			IF (tmrHorEntryNotPresent.q AND I_HOR_DnStream_Cv_Full) OR
				mc.DryRun THEN
				TimeoutTrigger 					:= FALSE;
				Station.RunStep	:= Station.RunStep + 10;
			END_IF

	40 : 	(************* Carton Send to Exit Conveyor  ****************)
			Station.Status 		:= '40: Carton Send to Exit Conveyor';
			Station.StatusInt	:= 354;
			
			IF NOT A_HOR_LC_Muting THEN
				HOR_BotCv_Mtr_Var.In_AutoON 			:= 	FALSE;
				HOR_TopCv_Mtr_Var.In_AutoON 			:= 	FALSE;


			(*	Case Counter *)				
					Statistic_CurShift_CaseProduce		:= Statistic_CurShift_CaseProduce + 1;
					Statistic_Total_CaseProduce			:= Statistic_Total_CaseProduce	+1;
					Statistic_Man_Total_CaseProduce		:= Statistic_Man_Total_CaseProduce +1;
					
			(* Update Statistic *)
			IF NOT mc.DryRun THEN
				IF NOT TapeReel_ActivatedL OR  W_HOR_TapeLRefill THEN
					Statistic_Current.RejectLeftTape	:= Statistic_Current.RejectLeftTape + 1;
					Statistic_Manual.RejectLeftTape		:= Statistic_Manual.RejectLeftTape + 1;
					Statistic_Total.RejectLeftTape		:= Statistic_Total.RejectLeftTape + 1;					
					E_CartonTapingErrL					:= TRUE;	
					Exit_Case_NG 						:= TRUE;
				
					
				ELSIF NOT TapeReel_ActivatedR OR W_HOR_TapeRRefill THEN
					Statistic_Current.RejectRightTape	:= Statistic_Current.RejectRightTape + 1;
					Statistic_Manual.RejectRightTape	:= Statistic_Manual.RejectRightTape + 1;
					Statistic_Total.RejectRightTape		:= Statistic_Total.RejectRightTape + 1;
					E_CartonTapingErrR					:= TRUE;	
					Exit_Case_NG 						:= TRUE;

					
				ELSIF 	H_CartonWeight < (CurrRecipe.rWeightTarget - CurrRecipe.rWeightTol) AND Cfg_EnbWeightCheck THEN
					Statistic_Current.RejectUnderWeight	:= Statistic_Current.RejectUnderWeight	+ 1;
					Statistic_Manual.RejectUnderWeight	:= Statistic_Manual.RejectUnderWeight	+ 1;
					Statistic_Total.RejectUnderWeight	:= Statistic_Total.RejectUnderWeight	+ 1;
					Weight_Fail_Counter					:= Weight_Fail_Counter +1;
					Exit_Case_NG 						:= TRUE;
					
					
				ELSIF 	H_CartonWeight > (CurrRecipe.rWeightTarget + CurrRecipe.rWeightTol) AND Cfg_EnbWeightCheck THEN
					Statistic_Current.RejectOverWeight	:= Statistic_Current.RejectOverWeight + 1;
					Statistic_Manual.RejectOverWeight	:= Statistic_Manual.RejectOverWeight + 1;
					Statistic_Total.RejectOverWeight	:= Statistic_Total.RejectOverWeight + 1;
					Weight_Fail_Counter					:= Weight_Fail_Counter +1;
					Exit_Case_NG 						:= TRUE;

			
				ELSE
					Statistic_Current.GoodCase			:= Statistic_Current.GoodCase + 1;	
					Statistic_Manual.GoodCase			:= Statistic_Manual.GoodCase + 1;	
					Statistic_Total.GoodCase			:= Statistic_Total.GoodCase + 1;	
					Exit_Case_Good 						:= TRUE;
					Weight_Fail_Counter					:= 0;


				END_IF
				
			ELSE
					Statistic_Manual.GoodCase			:= Statistic_Manual.GoodCase + 1;
					Weight_Fail_Counter					:= 0;

			END_IF		
								
				Station.RunStep	:= Station.RunStep + 10;
			END_IF
	
	50: (************* Tilt In conveyor waiting for carton in position ****************)
			Station.Status 		:= '50: Tilt Conveyor Waiting For Carton In Position';
			
			HOR_Tilt_In_Mtr_Var.In_AutoON	:= TRUE;
			HOR_Tilt_Out_Mtr_Var.In_AutoON	:= TRUE;

			IF (TiltInCv_InPosDly.Q OR mc.DryRun) AND NOT I_HOR_Tilt_Out_Cv_Present  THEN	
				Station.RunStep	:= Station.RunStep + 10;
			END_IF	
				
	60: (************* Tilt Unit Tilt to Tilt Out Conveyor ****************)
			Station.Status 		:= '60: Tilt Unit Tilt Carton To Out Conveyor';
			
			EX_Tilt_Srv_Var.In_PosCmd := 85.0;
			EX_Tilt_Srv_Var.In_VelCmd := 100;
			EX_Tilt_Srv_Var.In_MoveAbs := TRUE; 
	
			IF fcComparePos(CurrPos:= EX_Tilt_Srv_Var.Out_CurrPos, TargetPos:= EX_Tilt_Srv_Var.In_PosCmd, Tolerance := 0.5) THEN
				EX_Tilt_Srv_Var.In_MoveAbs := FALSE; 
				Station.RunStep	:= 10000;
			END_IF
			(*temporarily disable referencing*)
	
	70: (************* Tilt Unit Start Seaching for Sensor ****************)
			Station.Status 		:= '70: Tilt Unit Searching for Home Sensor';
		
			EX_Tilt_Srv_Var.In_SetAbsRef	:= TRUE;
	
			IF NOT EX_Tilt_Srv_Var.Out_Referenced THEN
				Station.RunStep	:= Station.RunStep + 10;
			END_IF
	80: (************* Tilt Unit Waiting for Home Sensor ****************)	
			Station.Status 		:= '80: Tilt Unit Waiting for Homing Complete';
			
			HOR_Tilt_In_Mtr_Var.In_AutoON		:= FALSE;
	
	
			IF  EX_Tilt_Srv_Var.Out_Referenced THEN
				EX_Tilt_Srv_Var.In_SetAbsRef	:= FALSE;
				Station.RunStep					:= 1000;
			END_IF
			
	1000 : 	(************* Process Done ****************)
			Station.Status 		:= '1000: Process Done';	
			Station.StatusInt	:= 499;
			M_StepRun 			:= FALSE;
			HMI.T_OneCycleRun 	:= FALSE;			
			Station.RunStep 	:= 0;
			H_ER_CtnGlueDone	:= FALSE;
			H_HOR_CtnWeightOK	:= FALSE;
			TimeoutTrigger 		:= FALSE;
	END_CASE

(* Tilt Out Conveyor Stop *)
IF TiltOutCv_StopDly.Q	THEN
	HOR_Tilt_Out_Mtr_Var.In_AutoON		:= FALSE;
END_IF

	

ELSE
	Station.RunStep := 0;
	
	IF Station.MajorFault OR Station.MinorFault THEN
		Station.Status 		:= 'Station Error';
		Station.StatusInt	:= 4;
	ELSIF Station.Origin THEN
		Station.Status 		:= 'Station In Origin';
		Station.StatusInt	:= 5;
	ELSIF NOT Station.OriginSchRun AND NOT MC.OriginSchRun THEN
		Station.Status 		:= 'Station Not In Origin';
		Station.StatusInt	:= 6;
	END_IF
END_IF

Station.Running := (Station.RunStep>0) OR (sc[4].RunStep >0) ;

END_PROGRAM

// ---- POUs/Horizontal/HOR_Origin.TcPOU
PROGRAM HOR_Origin
VAR_IN_OUT
	Station		:structStationCtrl;
END_VAR
VAR
	HOR_WA_Origin		:BOOL;
	pls_OriginSchRun	:R_trig;
	Timeout				:Ton;
	TmrCartonExit		:Ton;
	TimeoutTrigger		:BOOL;
	TimeoutSetting		:TIME;
	tmr_FullSensorDly	:TON;
	tmr_MtrStopped		:ton;
		
END_VAR

(**************************************************************************************************************)
(* Station Width Adjust in Origin Condition *)
(**************************************************************************************************************)
HOR_WA_Origin := 	TRUE ;

(**************************************************************************************************************)
(* Station Origin Condition *)
(**************************************************************************************************************)

Station.Origin 	:=	(
					(NOT I_HOR_Entry_Cv_Present OR H_ER_CtnGlueDone) AND
					HOR_BotCv_Mtr_Var.S_InvRdy AND
					HOR_TopCv_Mtr_Var.S_InvRdy AND
					HOR_WA_Origin AND
					EX_Tilt_Srv_Var.Out_Referenced AND
					tmr_MtrStopped.Q and
					Station.OriginRunStep =0)OR
					Station.Bypass;
					 		
(**************************************************************************************************************)
(* Individual Station Origin Run Trigger *)
(**************************************************************************************************************)
IF MC.ManualMode AND NOT Station.Origin AND NOT (Station.MajorFault OR Station.MinorFault OR MC.Trouble OR MC.StopPressed )  THEN
	IF Station.T_OriginSearch THEN
		Station.OriginSchRun  := TRUE;
	END_IF;
ELSE
	Station.OriginSchRun := FALSE;
	HOR.T_OriginSearch := FALSE;
END_IF;

(**************************************************************************************************************)
(* Station Origin Step *)
(**************************************************************************************************************)

Timeout(IN:=TimeoutTrigger, PT:=TimeoutSetting);
IF Timeout.Q THEN
	TimeoutTrigger := FALSE;
END_IF

pls_OriginSchRun(CLK:= (MC.OriginSchRun OR Station.OriginSchRun));
TmrCartonExit (in:= NOT I_HOR_DnStream_Cv_Full AND NOT I_HOR_Entry_Cv_Present  AND (Station.OriginRunStep = 30), pt:=T#10S);
tmr_FullSensorDly (IN:= (Station.OriginRunStep >= 30) AND I_HOR_DnStream_Cv_Full, PT:= T#3S);
tmr_MtrStopped( IN:= NOT HOR_BotCv_Mtr_Var.S_Running AND NOT HOR_TopCv_Mtr_Var.S_Running , pt:= T#2S);

IF (MC.OriginSchRun OR Station.OriginSchRun) AND NOT Station.Bypass  THEN
	CASE Station.OriginRunStep OF

	0 : 	(************* Ready To Run ****************)
			IF NOT Station.Origin AND pls_OriginSchRun.Q THEN
				Station.OriginRunStep := Station.OriginRunStep+10;	
			END_IF

	10	:	(************* Clear Tilt In and Tilt Out Conveyor ****************)
			Station.Status := 'Org10: Tilt Conveyor In and Out Run';
			
			HOR_Tilt_In_Mtr_Var.In_OrgOn	:= TRUE;
			HOR_Tilt_Out_Mtr_Var.In_OrgOn	:= TRUE;

			IF NOT I_HOR_Tilt_Out_Cv_Present THEN
				Station.OriginRunStep := Station.OriginRunStep+10;
			END_IF
			
	20:		(************ Tilt Unit Origin **********************)
			Station.Status := 'Org20: Tilt Servo Start to Home';
			
			EX_Tilt_Srv_Var.In_SetAbsRef	:= TRUE;
			
			IF NOT EX_Tilt_Srv_Var.Out_Referenced THEN
				Station.OriginRunStep	:= Station.OriginRunStep + 10;
			END_IF
	
	30: (***************** Waiting for Tilt Unit Origin Done ************)
			Station.Status := 'Org30: Tilt Servo Homing';
		
			IF  EX_Tilt_Srv_Var.Out_Referenced THEN
				EX_Tilt_Srv_Var.In_SetAbsRef	:= FALSE;
				Station.OriginRunStep	:= Station.OriginRunStep + 10;
			END_IF
		
	40 : 	(************* Cek Carton On Conveyor ****************)
			Station.Status := 'Org40: Cek Carton On Conveyor';
			HOR_BotCv_Mtr_Var.In_OrgOn	:= TRUE;
			HOR_TopCv_Mtr_Var.In_OrgOn	:= TRUE;
			EX_StpCylR_Var.In_OrgHome	:= TRUE;
			EX_StpCylL_Var.In_OrgHome	:= TRUE;
			
			IF I_HOR_Entry_Cv_Present THEN
				Station.Status := 'Org10: Top and Bottom Motor Run';
			ELSE
				Station.OriginRunStep := Station.OriginRunStep+10;
			END_IF
	
	50 : 	(************* Carton Send to Exit Conveyor  ****************)
			Station.Status 		:= 'Org50: Carton Send to Exit Conveyor';
			
			
			IF NOT I_HOR_Entry_Cv_Present THEN
				Station.OriginRunStep	:= Station.OriginRunStep + 10;
			END_IF

	60 : 	(************* Carton Send to Exit Conveyor  ****************)
			Station.Status 		:= 'Org60: Carton Send to Exit Conveyor';
			Station.StatusInt	:= 354;
			
			H_ER_CtnRdyForGlue	:=FALSE;
			H_ER_CtnGlueDone	:=FALSE;
			H_ER_CtnWeightOK	:=FALSE;				

			IF  tmr_FullSensorDly.Q OR TmrCartonExit.q THEN

				EX_StpCylR_Var.In_Orgwork	:= TRUE;
				EX_StpCylL_Var.In_Orgwork	:= TRUE;
				EX_StpCylR_Var.In_OrgHome	:= FALSE;
				EX_StpCylL_Var.In_OrgHome	:= FALSE;
				Station.OriginRunStep 		:= 40;
			END_IF

	70:	(******************** Make sure Conveyor is stopped **********************)
				HOR_BotCv_Mtr_Var.In_OrgOn 		:= FALSE;
				HOR_TopCv_Mtr_Var.In_OrgOn		:= FALSE;
				HOR_BotCv_Mtr_Var.T_ManOn 		:= FALSE;
				HOR_TopCv_Mtr_Var.T_ManOn		:= FALSE;	
				HOR_Tilt_In_Mtr_Var.In_OrgOn	:= FALSE;
				HOR_Tilt_Out_Mtr_Var.In_OrgOn	:= FALSE;				
			
		IF  tmr_MtrStopped.Q THEN
				Station.OriginRunStep 		:= 0;
			END_IF
		
	END_CASE

ELSE

	Station.OriginRunStep := 0;	

	
END_IF

END_PROGRAM

// ---- POUs/Horizontal/Option_90Deg_Conv.TcPOU
PROGRAM Option_90Deg_Conv
VAR
	bEnable			:BOOL;
	Full_Timer_ON	: TON;
	Clear_Timer_ON	: tOF;
	
END_VAR

bEnable := NOT MC.Trouble;
Full_Timer_ON	(IN:= I_HOR_DnStream_Cv_Full , PT:= T#2S);
Clear_Timer_ON	(IN:= I_HOR_90Deg_Full_PE, PT:= T#3S);

EX_Deg_Cyl_Var.In_HomeXLock := TRUE;
EX_Deg_Cyl_Var.In_WorkXLock := TRUE;

EX_90Deg_Cyl(				
	IN_CylName		:='TILT CV CYLINDER', 	
	In_Enable		:= Cfg_Exit90DegConv, 	
	In_Reset		:= MC.ResetPressed, 	
	In_WorkRS		:= I_HOR_90Deg_Tilt_Cly_Up, 	
	In_HomeRS		:= I_HOR_90Deg_Tilt_Cly_Dn, 	
	In_WorkTON		:= T#100MS, 	
	In_HomeTON		:= T#10MS, 	
	in_Timeout		:= T#5S, 	
	Out_WorkSV		=> O_HOR_90Deg_Cyl_Up, 	
	Out_HomeSV		=> O_HOR_90Deg_Cyl_Dn, 	
	CylVar			:= EX_Deg_Cyl_Var,
	Station			:= SC[6]);
	
(*	Control Condition	*)
IF 	SC[6].AutoRun			AND
	Full_Timer_ON.Q	AND
	not Clear_Timer_ON.q THEN
	EX_Deg_Cyl_Var.In_AutoWork	:= TRUE;
	EX_Deg_Cyl_Var.In_AutoHome	:= FALSE;
ELSE
	EX_Deg_Cyl_Var.In_AutoWork	:= FALSE;
	EX_Deg_Cyl_Var.In_AutoHome	:= TRUE;
END_IF

END_PROGRAM

// ---- POUs/Horizontal/HOR_Servo_Output.TcPOU
PROGRAM HOR_Servo_Output
VAR
	Reset:BOOL;
	bEnable:BOOL;
	plsStopMove: R_trig;
	debugcode: INT;
	debugcode2: INT;
END_VAR

IF (MC.AutoMode OR SC[6].M_Step) THEN
	EX_Tilt_Srv_Var.In_ServoOn := TRUE;
END_IF

IF HOR.OriginSchRun OR MC.OriginSchRun OR mc.AutoMode OR (mc.ResetPressed AND NOT mc.Trouble) THEN
	EX_Tilt_Srv_Var.In_ServoOn := TRUE;
END_IF

bEnable := NOT (SC[6].MajorFault OR MC.Trouble);

EX_Tilt_Srv_Var.In_MoveXLock := TRUE ;
EX_Tilt_Srv_Input.wSignalstatuswort.13	:= TRUE;
EX_Tilt_Srv_Input.wSignalstatuswort.14	:= TRUE;


EX_Tilt_Srv_Drive(
	In_Enable:= bEnable, 
	In_Reset := MC.ResetPressed,
	In_AbsEncoder:= FALSE, 
	In_DriveInput:= EX_Tilt_Srv_Input, 
	In_CommState:= EX_Tilt_Srv_State, 
	Out_DriveOutput=> EX_Tilt_Srv_Output, 
	Out_DriveFeedRateOverride=> , 
	DriveVar:= EX_Tilt_Srv_Var,
	Station			:= SC[6]);
	
IF mc.ManualMode THEN	
	EX_Tilt_Srv_Feedrate := 10000;
ELSE
	EX_Tilt_Srv_Feedrate :=    INT_TO_UINT(hmi.V_MachineSpeed * 100);
END_IF

END_PROGRAM

// ---- POUs/Horizontal/HOR_Motor_Output.TcPOU
PROGRAM HOR_Motor_Output
VAR
	Reset:BOOL;
	bEnable: BOOL;
	bManualReject	:BOOL;
	tmrManualReject	:Ton;
	bManualRejectNeg	:R_trig;
	
	
END_VAR

(******************** Error Stop ***********************)
IF E_Top_Conv_Jam or E_Bottom_Conv_Jam  THEN
	HOR_BotCv_Mtr_Var.E_OnErr	:= TRUE;
	HOR_TopCv_Mtr_Var.E_OnErr	:= TRUE;
END_IF
(********************************************************)

bEnable := NOT MC.Trouble AND Cfg_HorizontalExit;
HOR_BotCv_Mtr_Var.In_SpeedSel :=3;
HOR_BotCv_Mtr_Var.In_MoveXLock := TRUE;

HOR_BotCv_Mtr(
	IN_DevName:= 'HORIZON. BOTTOM CV', 
	In_Enable:= bEnable, 
	In_Reset:= MC.ResetPressed, 
	In_InvRdy := I_HOR_BotCv_InvRdy, 
	Out_InvRun => O_HOR_BotCv_Mtr_Run, 
	Out_InvDirc => O_HOR_BotCv_Mtr_Dirc, 
	Out_InvSpdBit0 => O_HOR_BotCv_Mtr_Spd1, 
	Out_InvSpdBit1 => O_HOR_BotCv_Mtr_Spd2,
	MotorVar:= HOR_BotCv_Mtr_Var,
	Station			:= SC[6]);


HOR_TopCv_Mtr_Var.In_MoveXLock := TRUE;
HOR_TopCv_Mtr_Var.In_SpeedSel :=3;
HOR_TopCv_Mtr(
	IN_DevName:= 'HORIZON. TOP CV', 
	In_Enable:= bEnable, 
	In_Reset:= MC.ResetPressed, 
	In_InvRdy := I_HOR_TopCv_InvRdy, 
	Out_InvRun => O_HOR_TopCv_Mtr_Run, 
	Out_InvDirc => O_HOR_TopCv_Mtr_Dirc, 
	Out_InvSpdBit0 => O_HOR_TopCv_Mtr_Spd1, 
	Out_InvSpdBit1 => O_HOR_TopCv_Mtr_Spd2,
	MotorVar:= HOR_TopCv_Mtr_Var,
	Station			:= SC[6]);


(* Reject Carton Manually *)	
tmrManualReject		(in:= bManualReject, pt:= T#10S);
bManualRejectNeg	( CLK := tmrManualReject.Q);

IF NOT tmrManualReject.Q AND bManualReject THEN
	HOR_TopCv_Mtr_Var.T_ManOn	:= TRUE;
	HOR_TopCv_Mtr_Var.T_ManOff	:= FALSE;
	WT_Mtr_Var.T_ManOn			:= TRUE;
	WT_Mtr_Var.T_ManOff			:= FALSE;
	HOR_BotCv_Mtr_Var.T_ManOn	:= TRUE;
	HOR_BotCv_Mtr_Var.T_ManOff	:= FALSE;	
	EX_FlapHoldL_Cyl_Var.T_ManHome	:= TRUE;
	EX_FlapHoldL_Cyl_Var.T_ManWork	:= FALSE;
	EX_FlapHoldR_Cyl_Var.T_ManHome	:= TRUE;
	EX_FlapHoldR_Cyl_Var.T_ManWork	:= FALSE;	
	Ex_SquarenessCylL_Var.T_ManHome	:= TRUE;
	Ex_SquarenessCylL_Var.T_ManWork	:= FALSE;
	Ex_SquarenessCylR_Var.T_ManHome	:= TRUE;
	Ex_SquarenessCylR_Var.T_ManWork	:= FALSE;	
	EX_StpCylL_Var.T_ManHome		:= TRUE;
	EX_StpCylL_Var.T_ManWork		:= FALSE;
	EX_StpCylR_Var.T_ManHome		:= TRUE;
	EX_StpCylR_Var.T_ManWork		:= FALSE;	
	
	IF 	H_ER_CtnRdyForGlue OR H_ER_CtnGlueDone OR H_ER_CtnWeightOK THEN
		Statistic_Current.RejectCaseRemoved	:= Statistic_Current.RejectCaseRemoved + 1;
		Statistic_Manual.RejectCaseRemoved	:= Statistic_Manual.RejectCaseRemoved + 1;
		Statistic_Total.RejectCaseRemoved	:= Statistic_Total.RejectCaseRemoved + 1;
	END_IF
	
	HMI.T_ClearExitMem			:= TRUE;	
END_IF

IF bManualRejectNeg.Q  THEN
	HOR_TopCv_Mtr_Var.T_ManOn	:= FALSE;
	WT_Mtr_Var.T_ManOn			:= FALSE;
	HOR_BotCv_Mtr_Var.T_ManOn	:= FALSE;
	bManualReject				:= FALSE;
	HOR_TopCv_Mtr_Var.T_ManOff	:= TRUE;
	WT_Mtr_Var.T_ManOff			:= TRUE;
	HOR_BotCv_Mtr_Var.T_ManOff	:= TRUE;	
	HMI.T_ClearExitMem			:= FALSE;		
END_IF
(* Tilt In Conveyor *)
HOR_Tilt_In_Mtr_Var.In_MoveXLock := TRUE;
	
HOR_Tilt_In_Mtr(
	IN_DevName:= 'Tilt In CV', 
	In_Enable:= bEnable, 
	In_Reset:= MC.ResetPressed, 
	In_StarterOK:= TRUE, 
	Out_MotorOn=> O_HOR_TiltCV1_On, 
	MotorVar:= HOR_Tilt_In_Mtr_Var,
	Station			:= SC[6]);

(* Tilt Out Conveyor *)
HOR_Tilt_Out_Mtr_Var.In_MoveXLock := TRUE;
	
HOR_Tilt_Out_Mtr(
	IN_DevName:= 'Tilt Out CV', 
	In_Enable:= bEnable, 
	In_Reset:= MC.ResetPressed, 
	In_StarterOK:= TRUE, 
	Out_MotorOn=> O_HOR_TiltCV2_On, 
	MotorVar:= HOR_Tilt_Out_Mtr_Var,
	Station			:= SC[6]);

END_PROGRAM

// ---- POUs/MC/Track_and_Trace.TcPOU
PROGRAM Track_and_Trace
VAR
tmr_TnT_CrossPushToCase		: Tof;
tmr_TnT_CrossPushForward	: Tof;
tmr_TnT_CaseIndex			: Tof;	
tmr_TnT_GoodCaseDischarge	: Tof;


END_VAR

(* Case Format *)
(* 2.2.1	Case format *)
(* (for differentiation between 5000 and 10000 cases 0 for 5000 and 1 for 10000)*)
IF CurrRecipe.iStackY = 2 THEN
		O_TnT_CaseFormat	:= TRUE;
	ELSE
		O_TnT_CaseFormat	:= FALSE;	
END_IF

(* Cross push to case initiated *)
(* 2.2.2	Cross push to case initiated (signal to go high as cross push starts) *)
tmr_TnT_CrossPushToCase (IN:= SC[2].RunStep	= 10 , PT:= T#1S);
O_TnT_CrossPushToCase	:= tmr_TnT_CrossPushToCase.Q;

(* Cross Push Fully Forward *)
(* 2.2.3	Cross push fully forward (Outers pushed into case- signal to go high)*)
tmr_TnT_CrossPushForward (IN:= SC[2].RunStep	= 110 , PT:= T#1S);
O_TnT_CrossPushForward	:= tmr_TnT_CrossPushForward.Q;

(* Case Index *)
(* 2.2.4	Case index (as machine indexes signal to go high at start of index)*)
tmr_TnT_CaseIndex	(IN:= SC[3].RunStep	= 30 , PT:= T#1S);
O_TnT_CaseIndex			:= tmr_TnT_CaseIndex.Q;

(* Good Case Discharge *)
(* 2.2.5	Good case discharged (i.e. signal high if case is not to be rejected – on as case exits machine)*)
tmr_TnT_GoodCaseDischarge	(IN:= Exit_Case_Good , PT:= T#1S);
O_TnT_GoodCaseDischarge		:= tmr_TnT_GoodCaseDischarge.Q;

END_PROGRAM

// ---- POUs/MC/Memory_Handling.TcPOU
PROGRAM Memory_Handling
VAR
	plsMemoryReset: R_trig;
	plsPurgeErectorCaseOff: R_trig;
	T_ManPurge: INT;
	tmrPurgeErectorCase:tof;
END_VAR

plsMemoryReset(CLK:=MC.DryRun);

IF plsMemoryReset.Q OR HMI.T_ClearAllMem OR MC_WA_Run THEN
	H_CO_StkRdyForXPush:=FALSE;
	H_CO_StkRdyForYPush:=FALSE;	
	H_ER_CtnRdyForPushIn:=FALSE;
	H_ER_CtnPushInDone:=FALSE;
	H_ER_CtnSideFlapDone:=FALSE;
	H_ER_CtnRdyForGlue:=FALSE;
	H_ER_CtnGlueDone:=FALSE;
	H_ER_CtnWeightOK:=FALSE;
	H_EL_CtnTapeDone:=FALSE;
	H_EL_CtnWeightOK:=FALSE;
	H_CO_Bdl_StkY_Count := 0;
	H_CO_Bdl_StkZ_Count := 0;
END_IF

IF HMI.T_ClearCollatorMem THEN
	H_CO_StkRdyForXPush:=FALSE;
	H_CO_Bdl_StkZ_Count := 0;	
END_IF

IF HMI.T_ClearBufferMem THEN
	H_CO_StkRdyForYPush:=FALSE;	
	H_CO_Bdl_StkY_Count := 0;
END_IF

IF HMI.T_ClearErectorMem THEN
	H_ER_CtnRdyForPushIn:=FALSE;
	H_ER_CtnPushInDone:=FALSE;
	H_ER_CtnSideFlapDone:=FALSE;
END_IF

IF HMI.T_ClearExitMem THEN
	H_ER_CtnRdyForGlue:=FALSE;
	H_ER_CtnGlueDone:=FALSE;
	H_ER_CtnWeightOK:=FALSE;	
END_IF

IF HMI.T_ClearElevatorMem THEN
	H_EL_CtnTapeDone:=FALSE;
	H_EL_CtnWeightOK:=FALSE;
	H_HOR_CtnWeightOK:=FALSE;	
END_IF


tmrPurgeErectorCase ( IN:= HMI.T_PurgeErectorCase, pt:=T#1S);
plsPurgeErectorCaseOff(CLK:= NOT tmrPurgeErectorCase.q);

IF tmrPurgeErectorCase.Q THEN
	ER_BFlapL_Vac_Var.T_ManPurge 	:= TRUE;
	(*ER_BFlapR_Vac_Var.T_ManPurge 	:= TRUE;*)
	ER_Arm_Vac_Var.T_ManPurge 		:= TRUE;
	ER_FFlapR_Cyl_Var.T_ManHome 	:= TRUE;
	ER_RFlapR_Cyl_Var.T_ManHome 	:= TRUE;
	(*ER_BFlapR_Vac_Var.T_ManPurge 	:= TRUE;*)
	ER_BFlapL_Vac_Var.T_ManPurge 	:= TRUE;
	ER_TFlapOpnL_Cyl_var.T_ManHome	:= TRUE;
	ER_TFlapClsL_Cyl_var.T_ManHome	:= TRUE;
	ER_TFlapOpnR_Cyl_var.T_ManHome	:= TRUE;
	ER_TFlapClsR_Cyl_var.T_ManHome	:= TRUE;
	ER_CaseGuideL_Cyl_Var.T_ManHome	:= TRUE;
	ER_CaseGuideR_Cyl_Var.T_ManHome	:= TRUE;
	H_ER_CtnRdyForPushIn			:=FALSE;
	H_ER_CtnPushInDone				:=FALSE;
	H_ER_CtnSideFlapDone			:=FALSE;
	
	IF H_ER_CtnErected	THEN
		Statistic_Current.RejectCaseRemoved	:= Statistic_Current.RejectCaseRemoved + 1;
		Statistic_Manual.RejectCaseRemoved	:= Statistic_Manual.RejectCaseRemoved + 1;
		Statistic_Total.RejectCaseRemoved	:= Statistic_Total.RejectCaseRemoved + 1;
	END_IF
	H_ER_CtnErected							:= FALSE;	
	
ELSIF plsPurgeErectorCaseOff.Q THEN
	ER_BFlapL_Vac_Var.T_ManPurge 	:= FALSE;
	(*ER_BFlapR_Vac_Var.T_ManPurge 	:= FALSE;*)
	ER_Arm_Vac_Var.T_ManPurge 		:= FALSE;
	ER_FFlapR_Cyl_Var.T_ManHome 	:= FALSE;
	H_ER_CtnRdyForPushIn			:=FALSE;
	H_ER_CtnPushInDone				:=FALSE;
	H_ER_CtnSideFlapDone			:=FALSE;	
END_IF

END_PROGRAM

// ---- POUs/FB/fbCylinderCtrl.TcPOU
FUNCTION_BLOCK fbCylinderCtrl

VAR_INPUT
	IN_CylName:STRING;
	In_Enable:BOOL;
	In_Reset:BOOL;
	(*Sensors*)
	In_WorkRS:BOOL;
	In_HomeRS:BOOL;	
	(*Timer*)
	In_WorkTON:TIME;
	In_HomeTON:TIME;
	in_Timeout:TIME;
END_VAR

VAR_OUTPUT
	Out_WorkSV:BOOL;
	Out_HomeSV:BOOL;	
END_VAR

VAR_IN_OUT
	CylVar:structCylinder;
	Station:structStationCtrl;
END_VAR

VAR

	Loc_Work:BOOL;
	Loc_Home:BOOL;
	Err_Cyl:BOOL;
	Fwd_TOut: TON;
	Bwd_TOut: TON;
	Fwd_TON: TON;
	Bwd_TON: TON;
	Loc_WorkPls: BOOL;
	FwdPls: R_TRIG;
	BwdPls: R_TRIG;
	Loc_HomePls: BOOL;
	Out_RSErr:BOOL;
	FwdPosPls: F_TRIG;
	BwdPosPls: F_TRIG;
END_VAR
VAR // added by the converter: edge detectors and wires of the graphical bodies
    _w1, _w2, _w3, _w4, _w5 : BOOL;
END_VAR

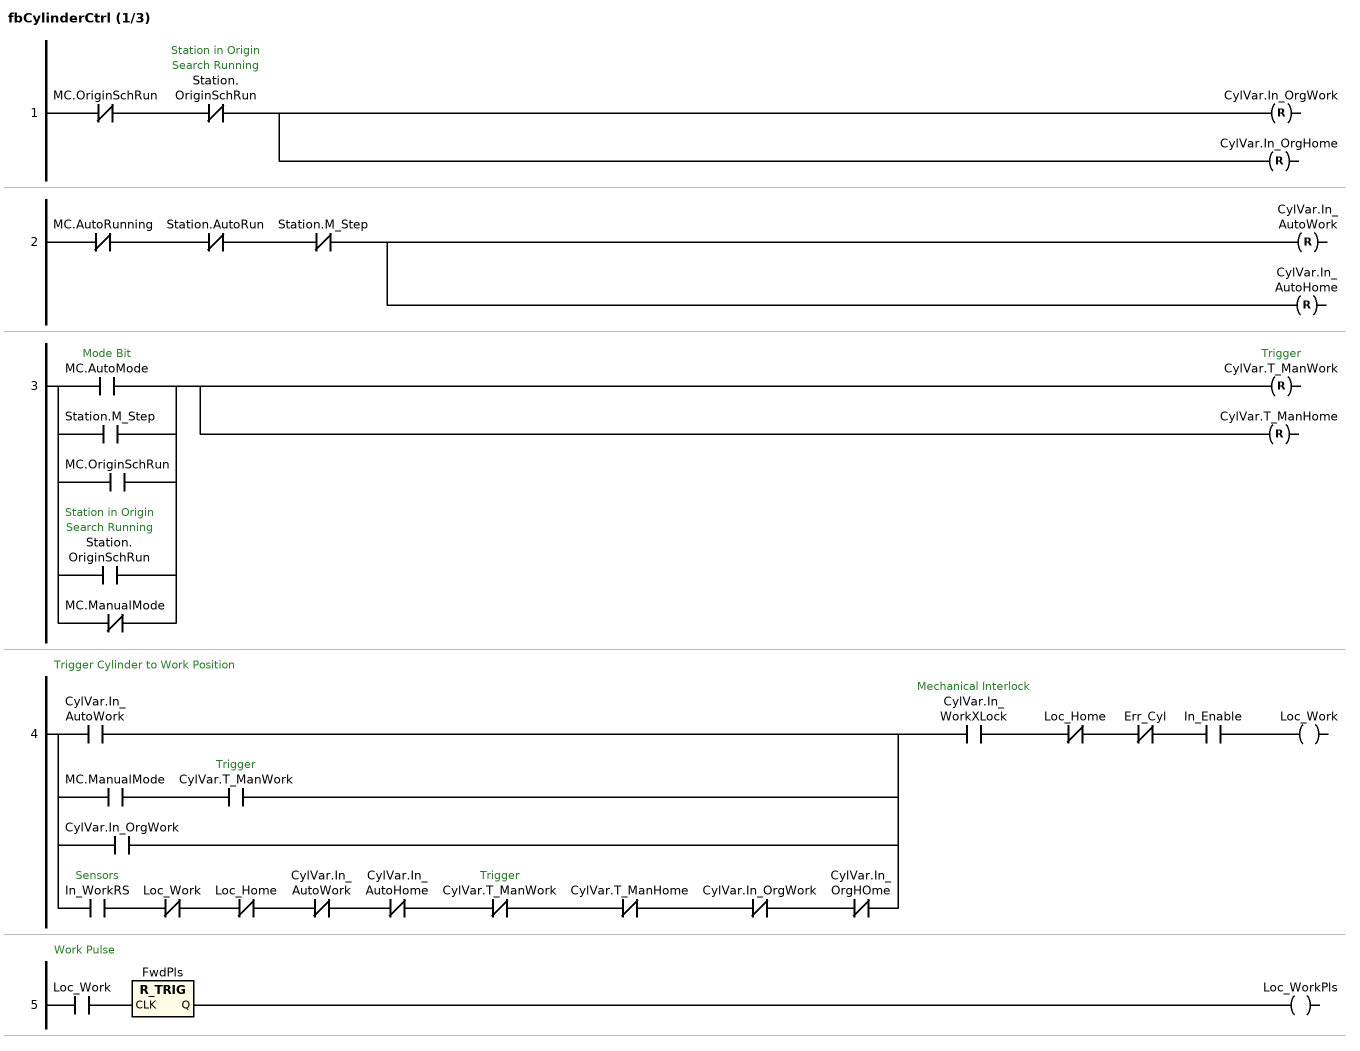
// NETWORK 1
//   Station.OriginSchRun: Station in Origin Search Running
_w1 := NOT MC.OriginSchRun AND NOT Station.OriginSchRun;
CylVar.In_OrgWork R= _w1;
CylVar.In_OrgHome R= _w1;

// NETWORK 2
_w2 := NOT MC.AutoRunning AND NOT Station.AutoRun AND NOT Station.M_Step;
CylVar.In_AutoWork R= _w2;
CylVar.In_AutoHome R= _w2;

// NETWORK 3
//   MC.AutoMode: Mode Bit
//   Station.OriginSchRun: Station in Origin Search Running
//   CylVar.T_ManWork: Trigger
_w3 := MC.AutoMode OR Station.M_Step OR MC.OriginSchRun OR Station.OriginSchRun OR NOT MC.ManualMode;
CylVar.T_ManWork R= _w3;
CylVar.T_ManHome R= _w3;

// NETWORK 4
// Trigger Cylinder to Work Position
//   CylVar.T_ManWork: Trigger
//   In_WorkRS: Sensors
//   CylVar.In_WorkXLock: Mechanical Interlock
Loc_Work := (CylVar.In_AutoWork OR MC.ManualMode AND CylVar.T_ManWork OR CylVar.In_OrgWork OR In_WorkRS AND NOT Loc_Work AND NOT Loc_Home AND NOT CylVar.In_AutoWork AND NOT CylVar.In_AutoHome AND NOT CylVar.T_ManWork AND NOT CylVar.T_ManHome AND NOT CylVar.In_OrgWork AND NOT CylVar.In_OrgHOme) AND CylVar.In_WorkXLock AND NOT Loc_Home AND NOT Err_Cyl AND In_Enable;

// NETWORK 5
// Work Pulse
FwdPls(CLK := Loc_Work); // R_TRIG
Loc_WorkPls := FwdPls.Q;

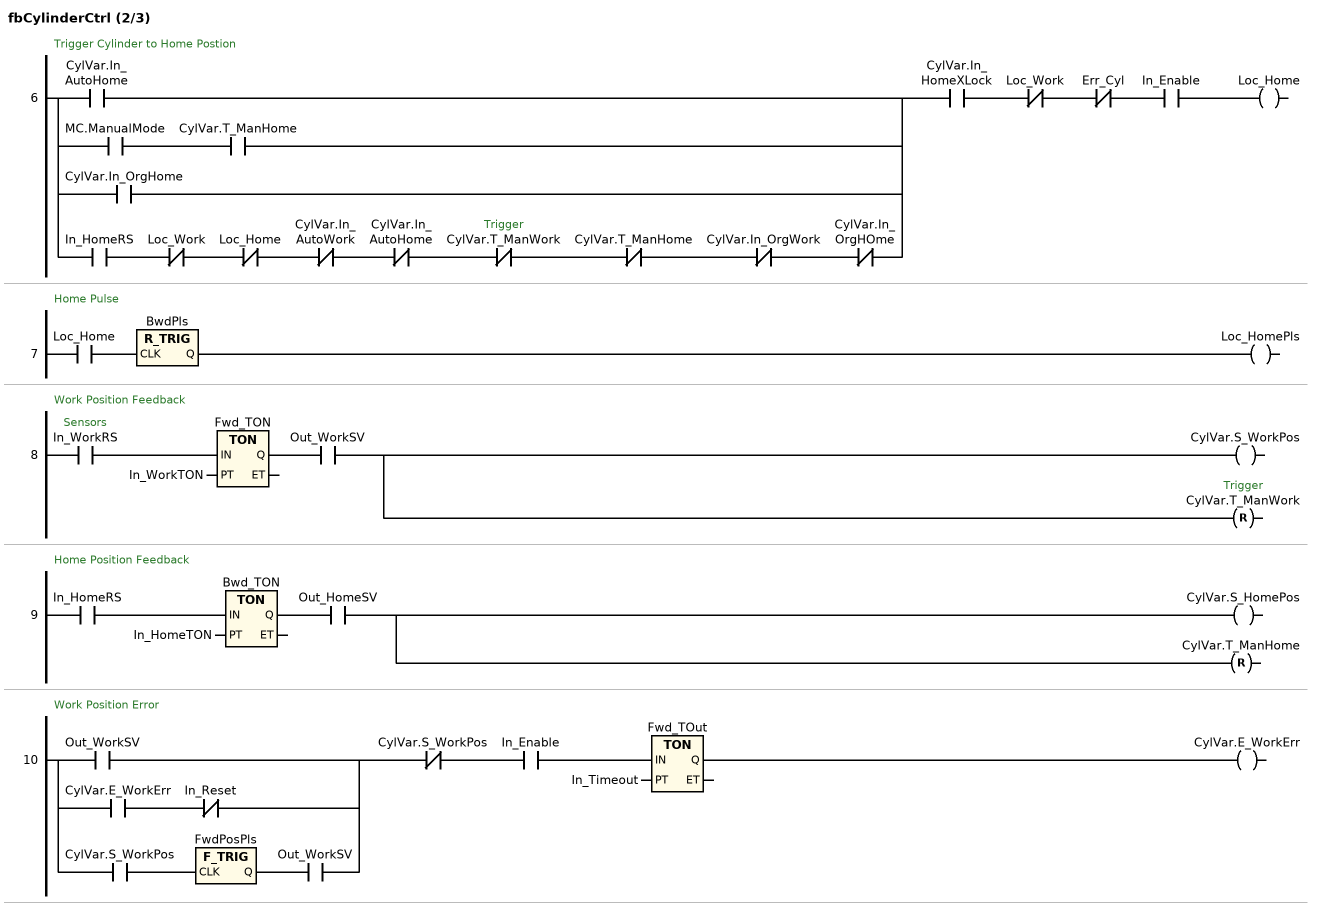
// NETWORK 6
// Trigger Cylinder to Home Postion
//   CylVar.T_ManWork: Trigger
Loc_Home := (CylVar.In_AutoHome OR MC.ManualMode AND CylVar.T_ManHome OR CylVar.In_OrgHome OR In_HomeRS AND NOT Loc_Work AND NOT Loc_Home AND NOT CylVar.In_AutoWork AND NOT CylVar.In_AutoHome AND NOT CylVar.T_ManWork AND NOT CylVar.T_ManHome AND NOT CylVar.In_OrgWork AND NOT CylVar.In_OrgHOme) AND CylVar.In_HomeXLock AND NOT Loc_Work AND NOT Err_Cyl AND In_Enable;

// NETWORK 7
// Home Pulse
BwdPls(CLK := Loc_Home); // R_TRIG
Loc_HomePls := BwdPls.Q;

// NETWORK 8
// Work Position Feedback
//   In_WorkRS: Sensors
//   In_WorkTON: Timer
//   CylVar.T_ManWork: Trigger
Fwd_TON(IN := In_WorkRS, PT := In_WorkTON); // TON
_w4 := Fwd_TON.Q AND Out_WorkSV;
CylVar.S_WorkPos := _w4;
CylVar.T_ManWork R= _w4;

// NETWORK 9
// Home Position Feedback
Bwd_TON(IN := In_HomeRS, PT := In_HomeTON); // TON
_w5 := Bwd_TON.Q AND Out_HomeSV;
CylVar.S_HomePos := _w5;
CylVar.T_ManHome R= _w5;

// NETWORK 10
// Work Position Error
FwdPosPls(CLK := CylVar.S_WorkPos); // F_TRIG
Fwd_TOut(IN := (Out_WorkSV OR CylVar.E_WorkErr AND NOT In_Reset OR FwdPosPls.Q AND Out_WorkSV) AND NOT CylVar.S_WorkPos AND In_Enable, PT := In_Timeout); // TON
CylVar.E_WorkErr := Fwd_TOut.Q;

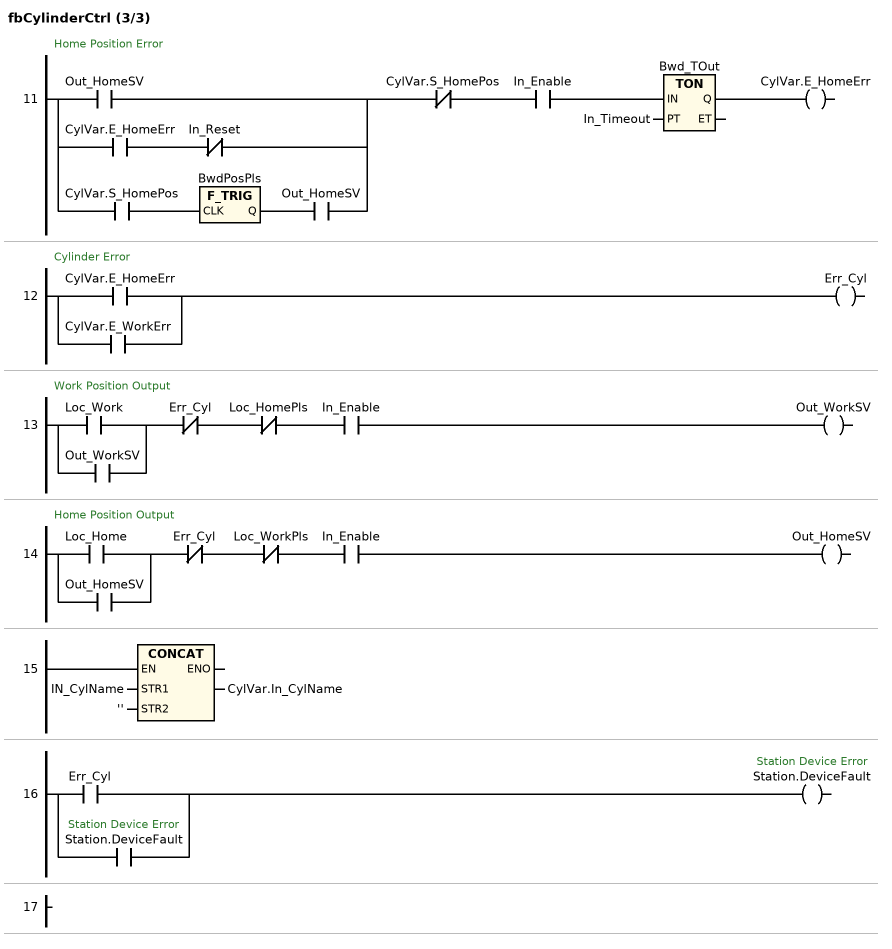
// NETWORK 11
// Home Position Error
BwdPosPls(CLK := CylVar.S_HomePos); // F_TRIG
Bwd_TOut(IN := (Out_HomeSV OR CylVar.E_HomeErr AND NOT In_Reset OR BwdPosPls.Q AND Out_HomeSV) AND NOT CylVar.S_HomePos AND In_Enable, PT := In_Timeout); // TON
CylVar.E_HomeErr := Bwd_TOut.Q;

// NETWORK 12
// Cylinder Error
Err_Cyl := CylVar.E_HomeErr OR CylVar.E_WorkErr;

// NETWORK 13
// Work Position Output
Out_WorkSV := (Loc_Work OR Out_WorkSV) AND NOT Err_Cyl AND NOT Loc_HomePls AND In_Enable;

// NETWORK 14
// Home Position Output
Out_HomeSV := (Loc_Home OR Out_HomeSV) AND NOT Err_Cyl AND NOT Loc_WorkPls AND In_Enable;

// NETWORK 15
CylVar.In_CylName := CONCAT(STR1 := IN_CylName, STR2 := '');

// NETWORK 16
//   Station.DeviceFault: Station Device Error
Station.DeviceFault := Err_Cyl OR Station.DeviceFault;

// NETWORK 17

END_FUNCTION_BLOCK

// ---- POUs/FB/fbCylinderCtrl_2Station.TcPOU
FUNCTION_BLOCK fbCylinderCtrl_2Station

VAR_INPUT
	IN_CylName:STRING;
	In_Enable:BOOL;
	In_Reset:BOOL;
	(*Sensors*)
	In_WorkRS:BOOL;
	In_HomeRS:BOOL;	
	(*Timer*)
	In_WorkTON:TIME;
	In_HomeTON:TIME;
	in_Timeout:TIME;
END_VAR

VAR_OUTPUT
	Out_WorkSV:BOOL;
	Out_HomeSV:BOOL;	
END_VAR

VAR_IN_OUT
	CylVar:structCylinder;
	Station:structStationCtrl;
	Station2:structStationCtrl;
END_VAR

VAR

	Loc_Work:BOOL;
	Loc_Home:BOOL;
	Err_Cyl:BOOL;
	Fwd_TOut: TON;
	Bwd_TOut: TON;
	Fwd_TON: TON;
	Bwd_TON: TON;
	Loc_WorkPls: BOOL;
	FwdPls: R_TRIG;
	BwdPls: R_TRIG;
	Loc_HomePls: BOOL;
	Out_RSErr:BOOL;
	FwdPosPls: F_TRIG;
	BwdPosPls: F_TRIG;
END_VAR
VAR // added by the converter: edge detectors and wires of the graphical bodies
    _w1, _w2, _w3, _w4, _w5 : BOOL;
END_VAR

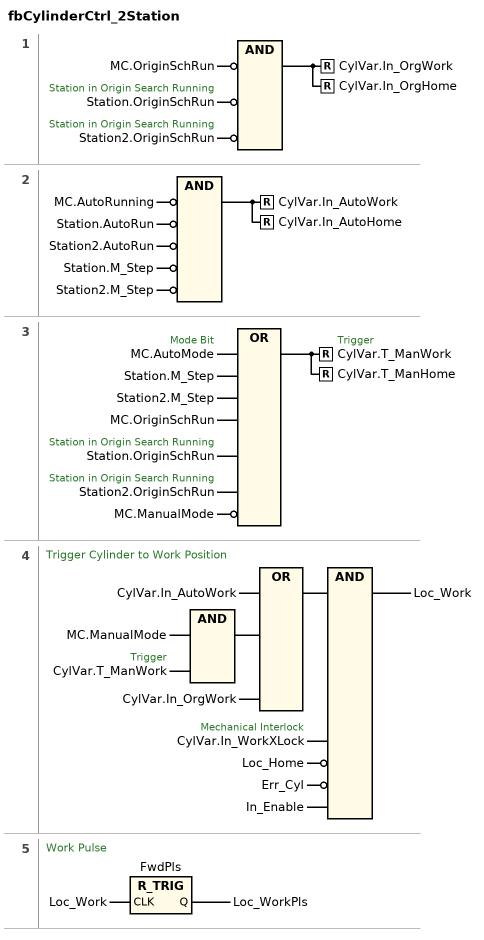
// NETWORK 1
//   Station.OriginSchRun: Station in Origin Search Running
//   Station2.OriginSchRun: Station in Origin Search Running
_w1 := NOT MC.OriginSchRun AND NOT Station.OriginSchRun AND NOT Station2.OriginSchRun;
CylVar.In_OrgWork R= _w1;
CylVar.In_OrgHome R= _w1;

// NETWORK 2
_w2 := NOT MC.AutoRunning AND NOT Station.AutoRun AND NOT Station2.AutoRun AND NOT Station.M_Step AND NOT Station2.M_Step;
CylVar.In_AutoWork R= _w2;
CylVar.In_AutoHome R= _w2;

// NETWORK 3
//   MC.AutoMode: Mode Bit
//   Station.OriginSchRun: Station in Origin Search Running
//   Station2.OriginSchRun: Station in Origin Search Running
//   CylVar.T_ManWork: Trigger
_w3 := MC.AutoMode OR Station.M_Step OR Station2.M_Step OR MC.OriginSchRun OR Station.OriginSchRun OR Station2.OriginSchRun OR NOT MC.ManualMode;
CylVar.T_ManWork R= _w3;
CylVar.T_ManHome R= _w3;

// NETWORK 4
// Trigger Cylinder to Work Position
//   CylVar.T_ManWork: Trigger
//   CylVar.In_WorkXLock: Mechanical Interlock
Loc_Work := (CylVar.In_AutoWork OR MC.ManualMode AND CylVar.T_ManWork OR CylVar.In_OrgWork) AND CylVar.In_WorkXLock AND NOT Loc_Home AND NOT Err_Cyl AND In_Enable;

// NETWORK 5
// Work Pulse
FwdPls(CLK := Loc_Work); // R_TRIG
Loc_WorkPls := FwdPls.Q;

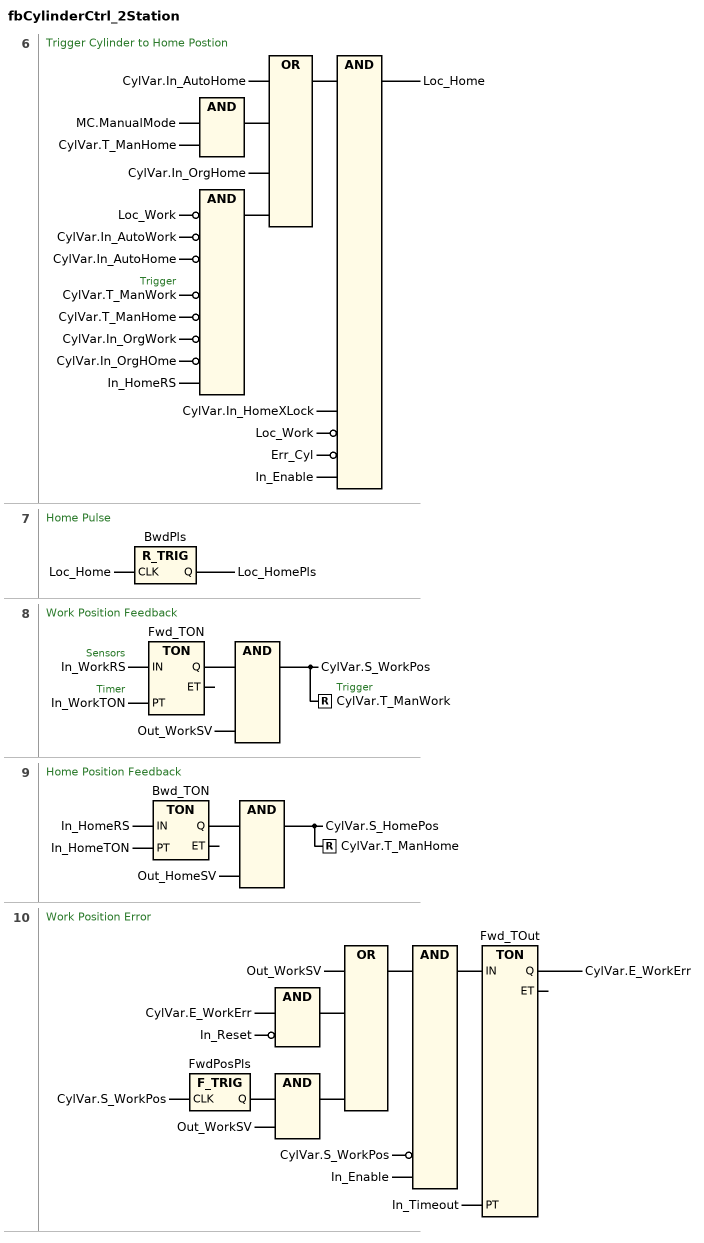
// NETWORK 6
// Trigger Cylinder to Home Postion
//   CylVar.T_ManWork: Trigger
Loc_Home := (CylVar.In_AutoHome OR MC.ManualMode AND CylVar.T_ManHome OR CylVar.In_OrgHome OR NOT Loc_Work AND NOT CylVar.In_AutoWork AND NOT CylVar.In_AutoHome AND NOT CylVar.T_ManWork AND NOT CylVar.T_ManHome AND NOT CylVar.In_OrgWork AND NOT CylVar.In_OrgHOme AND In_HomeRS) AND CylVar.In_HomeXLock AND NOT Loc_Work AND NOT Err_Cyl AND In_Enable;

// NETWORK 7
// Home Pulse
BwdPls(CLK := Loc_Home); // R_TRIG
Loc_HomePls := BwdPls.Q;

// NETWORK 8
// Work Position Feedback
//   In_WorkRS: Sensors
//   In_WorkTON: Timer
//   CylVar.T_ManWork: Trigger
Fwd_TON(IN := In_WorkRS, PT := In_WorkTON); // TON
_w4 := Fwd_TON.Q AND Out_WorkSV;
CylVar.S_WorkPos := _w4;
CylVar.T_ManWork R= _w4;

// NETWORK 9
// Home Position Feedback
Bwd_TON(IN := In_HomeRS, PT := In_HomeTON); // TON
_w5 := Bwd_TON.Q AND Out_HomeSV;
CylVar.S_HomePos := _w5;
CylVar.T_ManHome R= _w5;

// NETWORK 10
// Work Position Error
FwdPosPls(CLK := CylVar.S_WorkPos); // F_TRIG
Fwd_TOut(IN := (Out_WorkSV OR CylVar.E_WorkErr AND NOT In_Reset OR FwdPosPls.Q AND Out_WorkSV) AND NOT CylVar.S_WorkPos AND In_Enable, PT := In_Timeout); // TON
CylVar.E_WorkErr := Fwd_TOut.Q;

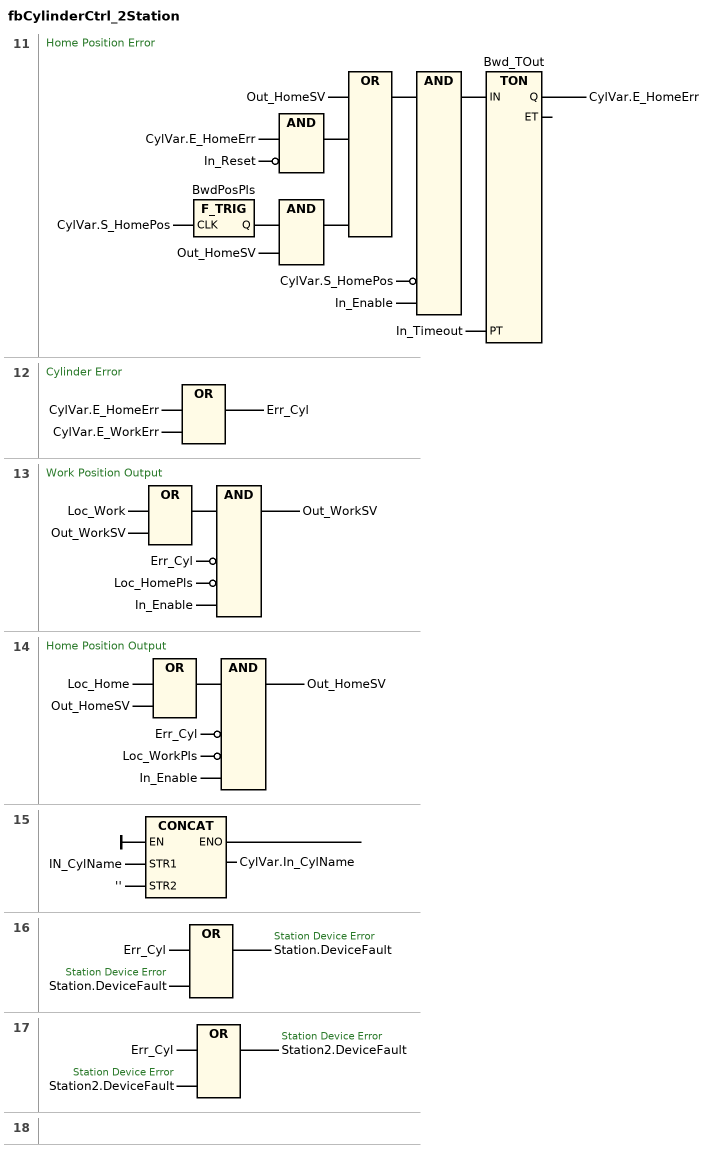
// NETWORK 11
// Home Position Error
BwdPosPls(CLK := CylVar.S_HomePos); // F_TRIG
Bwd_TOut(IN := (Out_HomeSV OR CylVar.E_HomeErr AND NOT In_Reset OR BwdPosPls.Q AND Out_HomeSV) AND NOT CylVar.S_HomePos AND In_Enable, PT := In_Timeout); // TON
CylVar.E_HomeErr := Bwd_TOut.Q;

// NETWORK 12
// Cylinder Error
Err_Cyl := CylVar.E_HomeErr OR CylVar.E_WorkErr;

// NETWORK 13
// Work Position Output
Out_WorkSV := (Loc_Work OR Out_WorkSV) AND NOT Err_Cyl AND NOT Loc_HomePls AND In_Enable;

// NETWORK 14
// Home Position Output
Out_HomeSV := (Loc_Home OR Out_HomeSV) AND NOT Err_Cyl AND NOT Loc_WorkPls AND In_Enable;

// NETWORK 15
CylVar.In_CylName := CONCAT(STR1 := IN_CylName, STR2 := '');

// NETWORK 16
//   Station.DeviceFault: Station Device Error
Station.DeviceFault := Err_Cyl OR Station.DeviceFault;

// NETWORK 17
//   Station2.DeviceFault: Station Device Error
Station2.DeviceFault := Err_Cyl OR Station2.DeviceFault;

// NETWORK 18

END_FUNCTION_BLOCK

// ---- POUs/FB/fbVacuumPumpCtrl.TcPOU
FUNCTION_BLOCK fbVacuumPumpCtrl

VAR_INPUT
	IN_DevName:STRING;
	In_Enable:BOOL;
	In_Reset:BOOL;

	(*Starter Healthy Signal*)
	In_StarterOK:BOOL;

END_VAR

VAR_OUTPUT
	Out_MotorOn:BOOL;

END_VAR

VAR_IN_OUT
	MotorVar:structMotorDirect;	
	Station:structStationCtrl;
END_VAR


VAR

	MotorOn:BOOL;
	On_TOut: TON;
	On_TON: TON;
	Loc_OnPls: BOOL;
	OnPls: R_TRIG;
	Out_RSErr:BOOL;
	OnPosPls: F_TRIG;

END_VAR

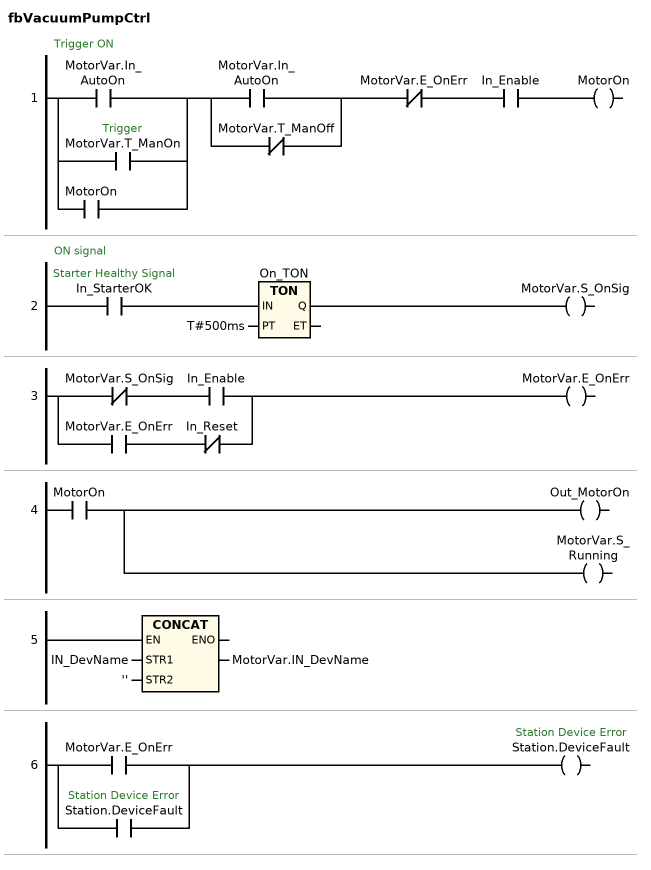
// NETWORK 1
// Trigger ON
//   MotorVar.T_ManOn: Trigger
MotorOn := (MotorVar.In_AutoOn OR MotorVar.T_ManOn OR MotorOn) AND (MotorVar.In_AutoOn OR NOT MotorVar.T_ManOff) AND NOT MotorVar.E_OnErr AND In_Enable;

// NETWORK 2
// ON signal
//   In_StarterOK: Starter Healthy Signal
On_TON(IN := In_StarterOK, PT := T#500ms); // TON
MotorVar.S_OnSig := On_TON.Q;

// NETWORK 3
MotorVar.E_OnErr := NOT MotorVar.S_OnSig AND In_Enable OR MotorVar.E_OnErr AND NOT In_Reset;

// NETWORK 4
Out_MotorOn := MotorOn;
MotorVar.S_Running := MotorOn;

// NETWORK 5
MotorVar.IN_DevName := CONCAT(STR1 := IN_DevName, STR2 := '');

// NETWORK 6
//   Station.DeviceFault: Station Device Error
Station.DeviceFault := MotorVar.E_OnErr OR Station.DeviceFault;

END_FUNCTION_BLOCK

// ---- POUs/FB/fbMotorDirectCtrl.TcPOU
FUNCTION_BLOCK fbMotorDirectCtrl

VAR_INPUT
	IN_DevName:STRING;
	In_Enable:BOOL;
	In_Reset:BOOL;

	(*Starter Healthy Signal*)
	In_StarterOK:BOOL;

END_VAR

VAR_OUTPUT
	Out_MotorOn:BOOL;

END_VAR

VAR_IN_OUT
	MotorVar:structMotorDirect;	
	Station:structStationCtrl;
END_VAR


VAR

	MotorOn:BOOL;
	On_TOut: TON;
	On_TON: TON;
	Loc_OnPls: BOOL;
	OnPls: R_TRIG;
	Out_RSErr:BOOL;
	OnPosPls: F_TRIG;

	pls_ManualModeOff: R_TRIG;
END_VAR

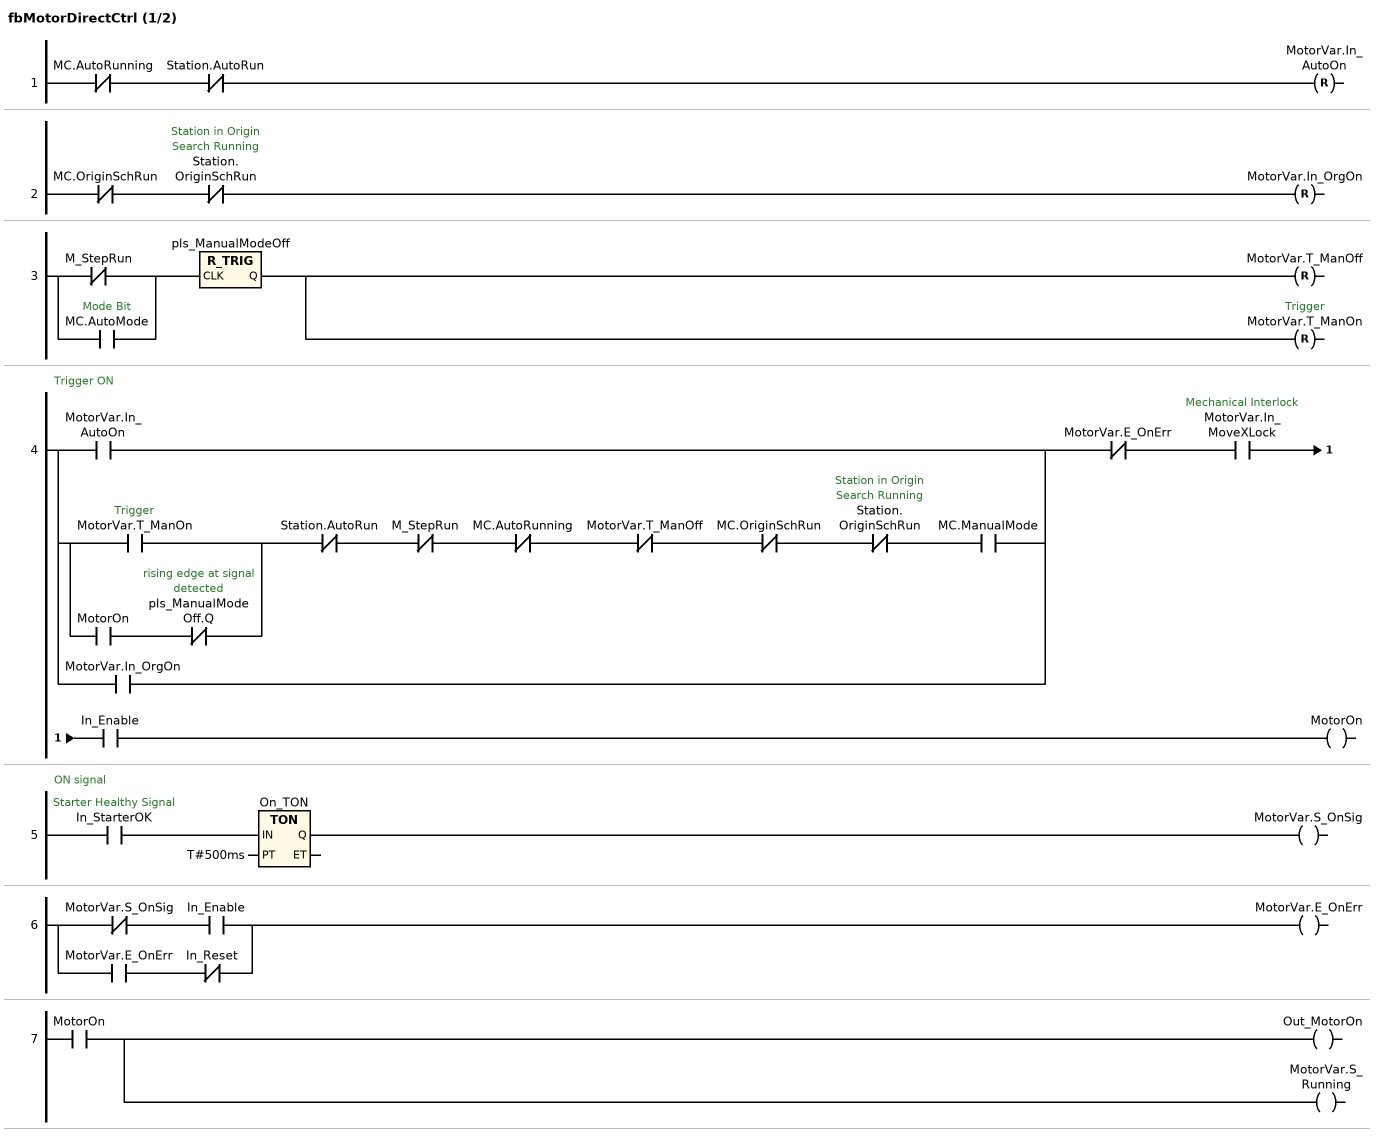
// NETWORK 1
MotorVar.In_AutoOn R= NOT MC.AutoRunning AND NOT Station.AutoRun;

// NETWORK 2
//   Station.OriginSchRun: Station in Origin Search Running
MotorVar.In_OrgOn R= NOT MC.OriginSchRun AND NOT Station.OriginSchRun;

// NETWORK 3
//   MC.AutoMode: Mode Bit
//   MotorVar.T_ManOn: Trigger
pls_ManualModeOff(CLK := NOT M_StepRun OR MC.AutoMode); // R_TRIG
MotorVar.T_ManOff R= pls_ManualModeOff.Q;
MotorVar.T_ManOn R= pls_ManualModeOff.Q;

// NETWORK 4
// Trigger ON
//   MotorVar.T_ManOn: Trigger
//   pls_ManualModeOff.Q: rising edge at signal detected
//   Station.OriginSchRun: Station in Origin Search Running
//   MotorVar.In_MoveXLock: Mechanical Interlock
MotorOn := (MotorVar.In_AutoOn OR (MotorVar.T_ManOn OR MotorOn AND NOT pls_ManualModeOff.Q) AND NOT Station.AutoRun AND NOT M_StepRun AND NOT MC.AutoRunning AND NOT MotorVar.T_ManOff AND NOT MC.OriginSchRun AND NOT Station.OriginSchRun AND MC.ManualMode OR MotorVar.In_OrgOn) AND NOT MotorVar.E_OnErr AND MotorVar.In_MoveXLock AND In_Enable;

// NETWORK 5
// ON signal
//   In_StarterOK: Starter Healthy Signal
On_TON(IN := In_StarterOK, PT := T#500ms); // TON
MotorVar.S_OnSig := On_TON.Q;

// NETWORK 6
MotorVar.E_OnErr := NOT MotorVar.S_OnSig AND In_Enable OR MotorVar.E_OnErr AND NOT In_Reset;

// NETWORK 7
Out_MotorOn := MotorOn;
MotorVar.S_Running := MotorOn;

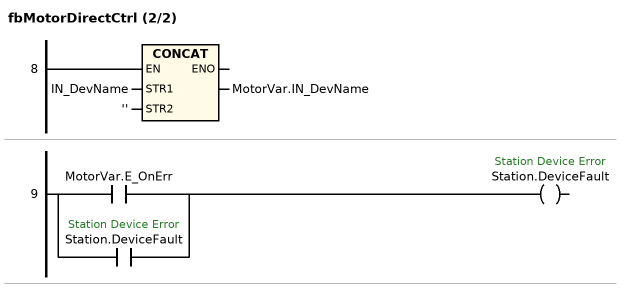
// NETWORK 8
MotorVar.IN_DevName := CONCAT(STR1 := IN_DevName, STR2 := '');

// NETWORK 9
//   Station.DeviceFault: Station Device Error
Station.DeviceFault := MotorVar.E_OnErr OR Station.DeviceFault;

END_FUNCTION_BLOCK

// ---- POUs/FB/fbMotorInverterCtrl.TcPOU
FUNCTION_BLOCK fbMotorInverterCtrl

VAR_INPUT
	IN_DevName:STRING;
	In_Enable:BOOL;
	In_Reset:BOOL;

	(*Inverter Healthy Signal*)
	In_InvRdy:BOOL;

END_VAR

VAR_OUTPUT
	Out_InvRun:BOOL;
	Out_InvDirc:BOOL;
	Out_InvSpdBit0:BOOL;
	Out_InvSpdBit1:BOOL;

END_VAR

VAR_IN_OUT
	MotorVar:structMotorInverter;	
	Station:structStationCtrl;
END_VAR


VAR

	MotorOn:BOOL;
	On_TOut: TON;
	On_TON: TON;
	NotRdy_TON:	TON;
	Loc_OnPls: BOOL;
	OnPls: R_TRIG;
	Out_RSErr:BOOL;
	OnPosPls: F_TRIG;
	TempInt:INT;

	pls_ManualModeOff: R_trig;
END_VAR

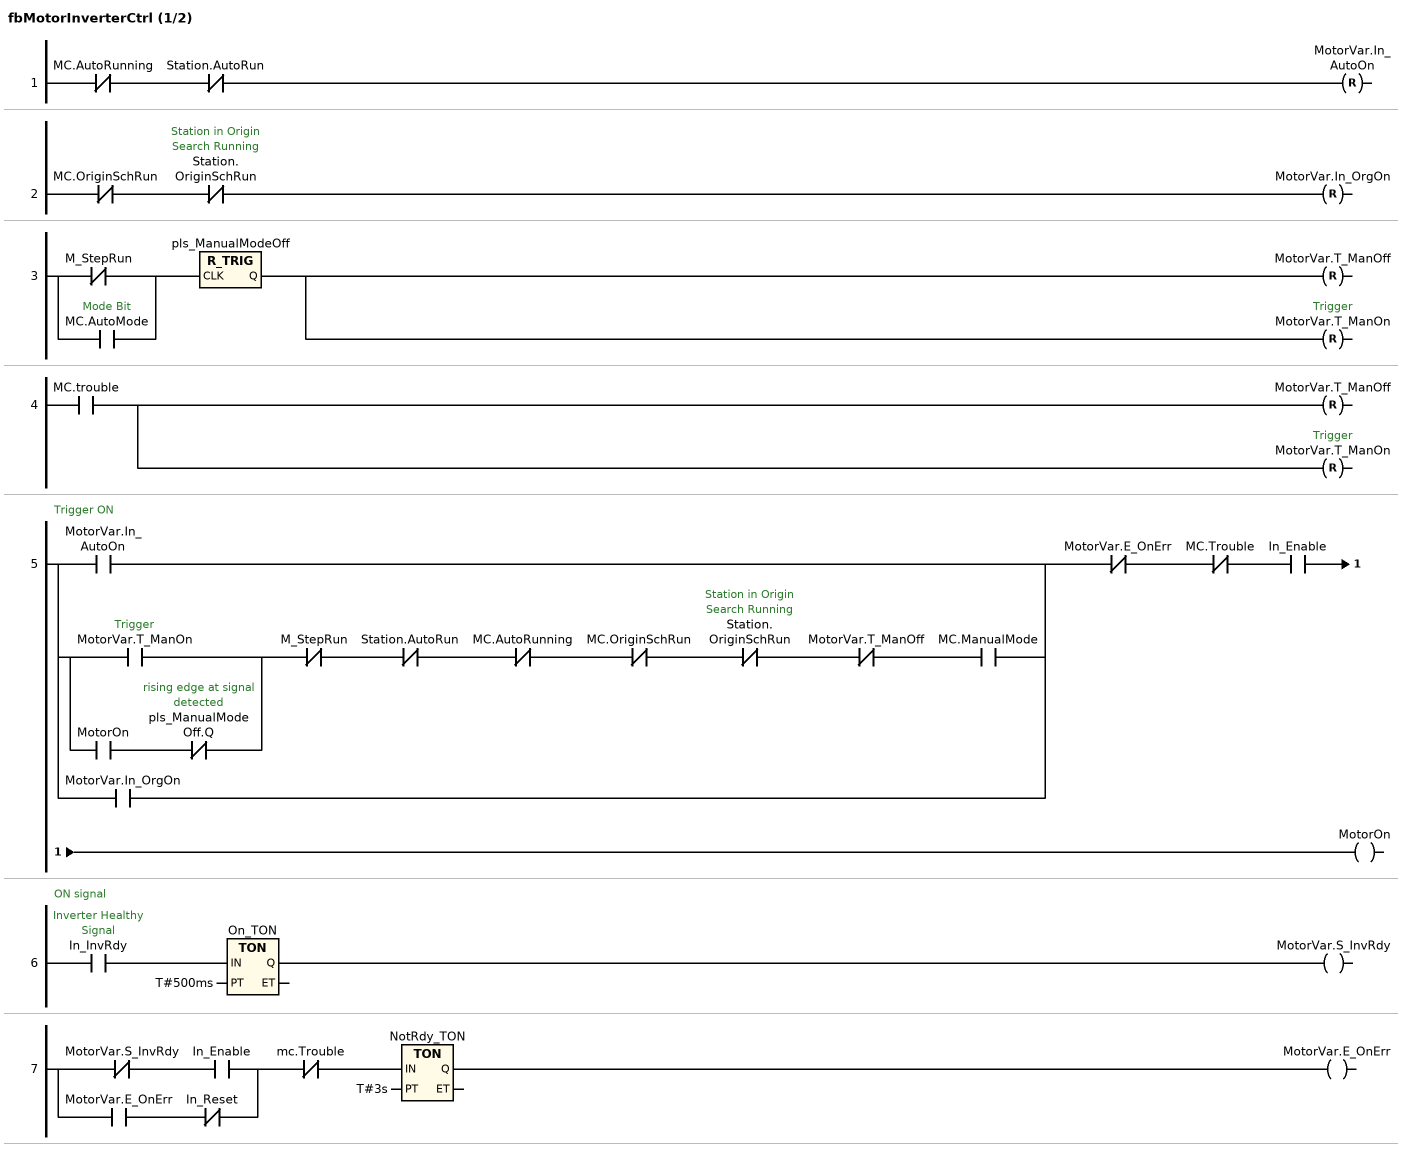
// NETWORK 1
MotorVar.In_AutoOn R= NOT MC.AutoRunning AND NOT Station.AutoRun;

// NETWORK 2
//   Station.OriginSchRun: Station in Origin Search Running
MotorVar.In_OrgOn R= NOT MC.OriginSchRun AND NOT Station.OriginSchRun;

// NETWORK 3
//   MC.AutoMode: Mode Bit
//   MotorVar.T_ManOn: Trigger
pls_ManualModeOff(CLK := NOT M_StepRun OR MC.AutoMode); // R_TRIG
MotorVar.T_ManOff R= pls_ManualModeOff.Q;
MotorVar.T_ManOn R= pls_ManualModeOff.Q;

// NETWORK 4
//   MotorVar.T_ManOn: Trigger
MotorVar.T_ManOff R= MC.trouble;
MotorVar.T_ManOn R= MC.trouble;

// NETWORK 5
// Trigger ON
//   MotorVar.T_ManOn: Trigger
//   pls_ManualModeOff.Q: rising edge at signal detected
//   Station.OriginSchRun: Station in Origin Search Running
MotorOn := (MotorVar.In_AutoOn OR (MotorVar.T_ManOn OR MotorOn AND NOT pls_ManualModeOff.Q) AND NOT M_StepRun AND NOT Station.AutoRun AND NOT MC.AutoRunning AND NOT MC.OriginSchRun AND NOT Station.OriginSchRun AND NOT MotorVar.T_ManOff AND MC.ManualMode OR MotorVar.In_OrgOn) AND NOT MotorVar.E_OnErr AND NOT MC.Trouble AND In_Enable;

// NETWORK 6
// ON signal
//   In_InvRdy: Inverter Healthy Signal
On_TON(IN := In_InvRdy, PT := T#500ms); // TON
MotorVar.S_InvRdy := On_TON.Q;

// NETWORK 7
NotRdy_TON(IN := (NOT MotorVar.S_InvRdy AND In_Enable OR MotorVar.E_OnErr AND NOT In_Reset) AND NOT mc.Trouble, PT := T#3s); // TON
MotorVar.E_OnErr := NotRdy_TON.Q;

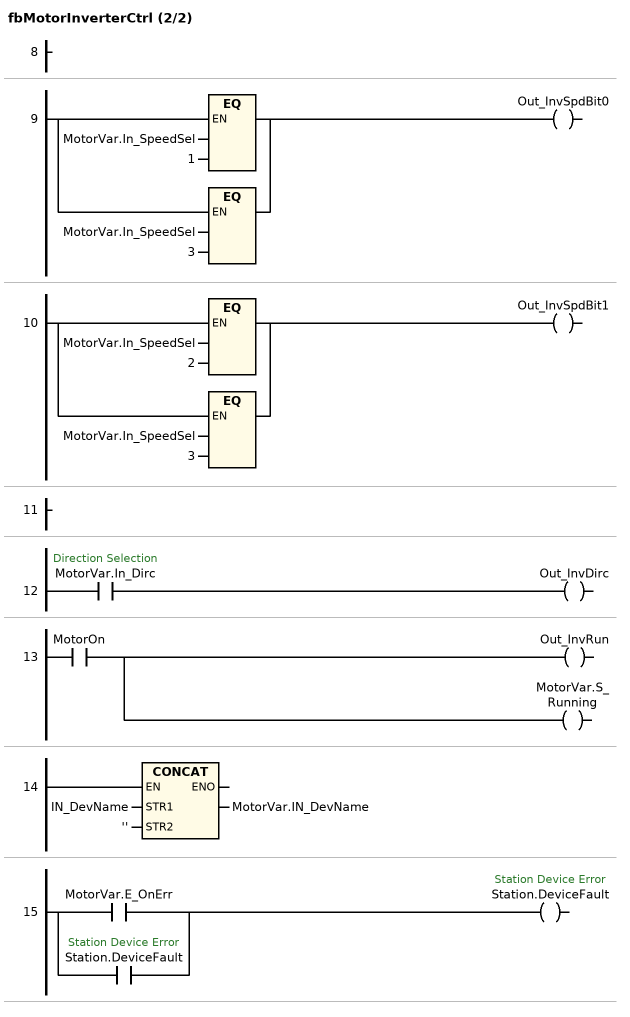
// NETWORK 8

// NETWORK 9
//   MotorVar.In_SpeedSel: Speed Selection 0-3
Out_InvSpdBit0 := MotorVar.In_SpeedSel = 1 OR MotorVar.In_SpeedSel = 3;

// NETWORK 10
//   MotorVar.In_SpeedSel: Speed Selection 0-3
Out_InvSpdBit1 := MotorVar.In_SpeedSel = 2 OR MotorVar.In_SpeedSel = 3;

// NETWORK 11

// NETWORK 12
//   MotorVar.In_Dirc: Direction Selection
Out_InvDirc := MotorVar.In_Dirc;

// NETWORK 13
Out_InvRun := MotorOn;
MotorVar.S_Running := MotorOn;

// NETWORK 14
MotorVar.IN_DevName := CONCAT(STR1 := IN_DevName, STR2 := '');

// NETWORK 15
//   Station.DeviceFault: Station Device Error
Station.DeviceFault := MotorVar.E_OnErr OR Station.DeviceFault;

END_FUNCTION_BLOCK

// ---- POUs/FB/fbIndradrive.TcPOU
FUNCTION_BLOCK PUBLIC fbIndradrive
VAR_INPUT
	In_Enable:BOOL;			(*1=Enable Drive, 0=Disable and ignore error*)
	In_Reset:BOOL;
	In_AbsEncoder:BOOL;		(*1=Absolute Encoder, 0=Incremental Encoder*)
	In_DriveInput:st_Indradrive_DCP_input ;		(*Indradrive Input Words via Ethercat*)
	In_CommState:UINT ;		(*Ethercat Slave State, 8=OK*)
	plsResetMode: R_trig;
END_VAR
VAR_OUTPUT
	Out_DriveOutput: st_Indradrive_DCP_output;	(*Indradrive Output Words via Ethercat*)
	Out_DriveFeedRateOverride: UINT;			(*Indradrive Output for Feedrate override, keep at 100%*)
END_VAR
VAR_IN_OUT
	DriveVar:structIndradrive;	(*Local Data structure to handle Indradrive variables*)
	Station:structStationCtrl;
END_VAR
VAR
	Drive: FB_Indradrive_DCP;	(*Standard Function Block Provided by Bosch*)
	tmrDriveEnableTOUT:TON;
	tmrHomingTOUT:TON;
	tmrMovePosTOUT:TON;
	tmrMajorErrorRecovery:Tof;
	diPosCmd:DINT;
	diVelCmd:DINT;
	DriveStatus:INT;
	plsInPos: R_TRIG;
	plsLimitTriggered: R_trig;
	plsMoveRel: R_trig;
	plsStopMove: R_TRIG;
	plsEMGReset: R_trig;
	ServoBusy:BOOL;
	plsMoveAbs: R_trig;
	plsStopMove2: R_trig;
	plsHomed: R_TRIG;
END_VAR
VAR CONSTANT
	FACTOR_DINT_REAL : INT := 10000;
	FACTOR_VEL_DINT_REAL : INT := 1000;
END_VAR

(* convert DINT values from FB to REAL values for the user program and vise versa*)
(* used only for trace purpose *)
DriveVar.Out_CurrPos := DINT_TO_REAL(Drive.diPOS_ACT) / FACTOR_DINT_REAL;
DriveVar.Out_CurrVel := DINT_TO_REAL(Drive.diVEL_ACT) / FACTOR_VEL_DINT_REAL;

(* REAL variables can be used for commanding instead of DINT variable used in the sample code *)
Drive.diPOS_CMD := REAL_TO_DINT (DriveVar.In_PosCmd * FACTOR_DINT_REAL);
Drive.diVEL_CMD := REAL_TO_DINT (DriveVar.In_VelCmd * FACTOR_VEL_DINT_REAL);

(*
(*Force Slow Speed in Manual Mode When close to Negative Limit For Accurate Referencing*)
IF DriveVar.Out_CurrPos <= 20 AND DriveVar.In_JogBwd THEN
	Drive.diVEL_CMD := 100 * FACTOR_VEL_DINT_REAL;
END_IF
*)

IF mc.ManualMode AND DriveVar.In_VelCmd > 1000 THEN
	DriveVar.In_VelCmd := 1000;
END_IF

Out_DriveFeedRateOverride := 100;

(***********************************************************************************************)
(*Servo Controller Status*)

IF NOT In_DriveInput.wSignalstatuswort.11 AND NOT In_DriveInput.wSignalstatuswort.12 THEN
	DriveStatus := 0;	(* Control section and power section not ready for operation (e.g., drive error or phase 2)*)
ELSIF NOT In_DriveInput.wSignalstatuswort.11 AND In_DriveInput.wSignalstatuswort.12 THEN
	DriveStatus := 1;	(* Control section ready for operation (bb)*)
ELSIF In_DriveInput.wSignalstatuswort.11 AND NOT In_DriveInput.wSignalstatuswort.12 THEN
	DriveStatus := 2;	(* Control section and power section ready for operation (Ab)*)
ELSIF In_DriveInput.wSignalstatuswort.11 AND In_DriveInput.wSignalstatuswort.12 THEN
	DriveStatus := 3;	(* Drive with torque (AF)*)
END_IF

(***********************************************************************************************)
(*Servo Limit Sensors Status*)
DriveVar.Out_PosLimit := In_DriveInput.wSignalstatuswort.13;
DriveVar.Out_NegLimit := In_DriveInput.wSignalstatuswort.14;

(***********************************************************************************************)
(*Error Handling*)

IF In_Reset THEN
	DriveVar.Out_ErrorWord := 0;
END_IF

Drive.bRESET := In_Reset;

(*Servo is in Alarm State Error*) 
IF Drive.bERROR AND In_Enable  THEN 
	DriveVar.Out_ErrorWord := 11;
END_IF

(*Servo Control and Power Section Not Ready Error*) 
IF DriveStatus = 0 AND In_Enable  THEN 
	DriveVar.Out_ErrorWord := 12;
END_IF

(*Servo Enable Timeout Error*) 
tmrDriveEnableTOUT(IN:= Drive.bDRIVE_ENABLE AND NOT (Drive.bQ_DRIVE_ENABLE AND Drive.bQ_MAIN_MODE),PT:=T#5S);
IF tmrDriveEnableTOUT.Q AND In_Enable THEN 
	DriveVar.Out_ErrorWord := 13;
END_IF

(*Servo Not Referenced Error*)
IF Drive.bQ_DRIVE_ENABLE AND NOT Drive.bIN_REFERENCE AND In_AbsEncoder AND In_Enable  THEN 
	DriveVar.Out_ErrorWord := 20;
END_IF

(*Servo Homing Timeout Error*) 
tmrHomingTOUT(IN:= Drive.bHOMING,PT:=T#300S);
IF tmrHomingTOUT.Q THEN 
	DriveVar.Out_ErrorWord := 21;
	Drive.bHOMING := FALSE;
END_IF

(*Servo Move Position Timeout Error*) 
tmrMovePosTOUT(IN:= (DriveVar.In_MoveAbs OR ServoBusy OR
					DriveVar.In_MoveRel) AND NOT DriveVar.Out_InPos,PT:=T#90S);
IF tmrMovePosTOUT.Q THEN 
	DriveVar.Out_ErrorWord := 22;
	ServoBusy := FALSE;
	DriveVar.In_MoveAbs := FALSE;
	DriveVar.In_MoveRel := FALSE;
END_IF

(*Servo Move Position Limit Error*) 
IF ServoBusy AND
	(((DriveVar.In_PosCmd < DriveVar.Out_CurrPos) AND NOT DriveVar.Out_NegLimit) 
	OR ((DriveVar.In_PosCmd > DriveVar.Out_CurrPos) AND NOT DriveVar.Out_PosLimit)) THEN 
	DriveVar.Out_ErrorWord := 23;
	ServoBusy := FALSE;
	DriveVar.In_MoveAbs := FALSE;
	DriveVar.In_MoveRel := FALSE;
END_IF

(*Servo Communication Error*) 
IF In_CommState <> 8 AND In_Enable  THEN
	DriveVar.Out_ErrorWord := 10;
END_IF

IF DriveVar.Out_ErrorWord > 1 THEN
	DriveVar.Out_Error := TRUE;
ELSE
	IF NOT DriveVar.In_MoveXLock THEN
		DriveVar.Out_ErrorWord := 0;
	ELSE
		DriveVar.Out_ErrorWord := 1;
	END_IF
	DriveVar.Out_Error := FALSE;
END_IF
(*Warning*)
DriveVar.Out_Warning := Drive.bWARNING;

(***********************************************************************************************)
(*Servo Enable*)

plsLimitTriggered(CLK:=NOT (DriveVar.Out_NegLimit AND DriveVar.Out_PosLimit));

IF plsLimitTriggered.Q THEN
	DriveVar.In_ServoOn := FALSE;
END_IF

IF In_Enable AND DriveVar.In_ServoOn AND NOT DriveVar.Out_Error
	AND DriveStatus >= 1 AND NOT Station.MinorFault  THEN
	(* drive enable and drive on commands *)
	Drive.bDRIVE_ENABLE:= TRUE;
	Drive.bDRIVE_START:= TRUE;
ELSE
	(* drive enable and drive on commands *)
	Drive.bDRIVE_ENABLE:= FALSE;
	Drive.bDRIVE_START:= FALSE;		
	DriveVar.Out_Busy := FALSE;
	DriveVar.In_JogBwd := FALSE;
	DriveVar.In_JogFwd := FALSE;
	DriveVar.In_MoveAbs := FALSE;
	DriveVar.In_MoveHome := FALSE;
	DriveVar.In_MoveRel := FALSE;
	DriveVar.In_ServoOn := FALSE;
END_IF

Drive.bIMMEDIATE_CHANGE := TRUE;
	
(***********************************************************************************************)
(*Servo Movement Control*)
(***********************************************************************************************)

(*Force Stop Command When Mode Changes*)
plsResetMode(CLK:= NOT MC.AutoMode);

plsStopMove(CLK:= NOT (Station.OriginSchRun OR MC.OriginSchRun OR 
						Station.AutoRun OR Station.M_Step));

plsStopMove2(CLK:= (Station.OriginSchRun OR MC.OriginSchRun OR
						Station.M_Step OR MC.AutoMode));
						
IF plsStopMove.Q AND plsStopMove2.Q OR plsResetMode.Q THEN
	DriveVar.In_StopMove := TRUE;
	DriveVar.In_MoveAbs := FALSE;
	DriveVar.In_MoveHome := FALSE;
	DriveVar.In_MoveRel := FALSE;
END_IF

(*Check New Move Command Direction for Interlocking Purpose*)
IF DriveVar.In_JogFwd OR 
	((DriveVar.In_PosCmd > DriveVar.Out_CurrPos) AND
		DriveVar.In_MoveAbs) OR
	((DriveVar.In_PosCmd > 0) AND
		DriveVar.In_MoveRel) THEN
	DriveVar.Out_PosDirc := TRUE;
	DriveVar.Out_NegDirc := FALSE;
ELSIF DriveVar.In_JogBwd OR 
	((DriveVar.In_PosCmd < DriveVar.Out_CurrPos) AND
		DriveVar.In_MoveAbs) OR
	((DriveVar.In_PosCmd < 0) AND
		DriveVar.In_MoveRel) THEN	
	DriveVar.Out_PosDirc := FALSE;
	DriveVar.Out_NegDirc := TRUE;
ELSE
	DriveVar.Out_PosDirc := FALSE;
	DriveVar.Out_NegDirc := FALSE;		
END_IF

IF Drive.bQ_DRIVE_ENABLE AND Drive.bQ_MAIN_MODE AND DriveStatus = 3 THEN
	DriveVar.Out_Ready := TRUE;
	
	(* Origin Search for Incremental Encoder Servo*)
	IF NOT In_AbsEncoder THEN		
		IF DriveVar.In_MoveHome AND NOT Drive.bIN_REFERENCE AND NOT DriveVar.Out_Busy
		AND Drive.diVEL_CMD > 0 THEN
			Drive.bHOMING := TRUE;
		END_IF
		IF Drive.bIN_REFERENCE THEN
			Drive.bHOMING := FALSE;
		END_IF
	END_IF
	
	(*Jog Command*)
	IF MC.ManualMode AND NOT Station.M_Step THEN
		IF DriveVar.In_JogFwd AND NOT DriveVar.In_JogBwd AND DriveVar.In_MoveXLock THEN
			(* Jog Positive command *)
			Drive.bJOG_FORWARD := TRUE;
			Drive.bJOG_BACKWARD := FALSE;
		ELSIF NOT DriveVar.In_JogFwd AND DriveVar.In_JogBwd AND DriveVar.In_MoveXLock THEN
			(* Jog Negative  command *)
			Drive.bJOG_FORWARD := FALSE;
			Drive.bJOG_BACKWARD := TRUE;
		ELSE
			(* Stop Jogging *)
			Drive.bJOG_FORWARD := FALSE;
			Drive.bJOG_BACKWARD := FALSE;
		END_IF
	ELSE
		DriveVar.In_JogFwd := FALSE;
		DriveVar.In_JogBwd := FALSE;
	END_IF
	
	IF Drive.bIN_REFERENCE THEN
		IF DriveVar.In_MoveXLock THEN
			(* Start Absolute move *)
			plsMoveAbs(CLK:=DriveVar.In_MoveAbs);
			IF DriveVar.In_MoveAbs AND Drive.bNEW_VALUE_POSSIBLE THEN
				ServoBusy := TRUE;
				(*DriveVar.In_MoveAbs := FALSE;*)
				IF Drive.diPOS_CMD <> Drive.diPOS_ACT AND Drive.diVEL_CMD <> 0 THEN
					DriveVar.Out_InPos := FALSE;
					Drive.bABS_REL := FALSE;       				(* False --> Absolute command *)
					IF Drive.bNEW_VALUE THEN
						Drive.bNEW_VALUE := FALSE;
					ELSE
						Drive.bNEW_VALUE := TRUE;
					END_IF
				END_IF
			END_IF
			(* Start Relative move *)
			plsMoveRel(CLK:=DriveVar.In_MoveRel);
			IF plsMoveRel.Q AND Drive.bNEW_VALUE_POSSIBLE AND 
				NOT ServoBusy  THEN
				ServoBusy := TRUE;
				DriveVar.In_MoveRel := FALSE;
				IF Drive.diPOS_CMD <> 0 AND Drive.diVEL_CMD <> 0 THEN
					DriveVar.Out_InPos := FALSE;
					Drive.bABS_REL := TRUE;       				(* True  --> Relative  command *)
					IF Drive.bNEW_VALUE THEN
						Drive.bNEW_VALUE := FALSE;
					ELSE
						Drive.bNEW_VALUE := TRUE;
					END_IF
				END_IF
			END_IF
		END_IF
	ELSE
		DriveVar.Out_InPos := FALSE;
	END_IF
	
	(*Set Servo Busy Status*)	
	DriveVar.Out_Busy := NOT Drive.bIN_STANDSTILL;
	IF DriveVar.Out_Busy THEN
		DriveVar.Out_InPos := FALSE; 
	END_IF
	
ELSE

	ServoBusy := FALSE;
	DriveVar.In_MoveAbs := FALSE;
	DriveVar.In_MoveRel := FALSE;
	DriveVar.Out_Ready := FALSE;
	DriveVar.In_JogBwd := FALSE;
	DriveVar.In_JogFwd := FALSE;
	DriveVar.In_MoveHome := FALSE;
	Drive.bJOG_FORWARD := FALSE;
	Drive.bJOG_BACKWARD := FALSE;
	Drive.bHOMING := FALSE;
	
END_IF

(* wait for InPos *)
plsInPos(CLK:= Drive.bPOS_OK);
plsEMGReset(CLK:= NOT MC.Trouble );
IF Drive.bPOS_OK AND 
	fcComparePos(CurrPos:= DriveVar.In_PosCmd, TargetPos:= DriveVar.Out_CurrPos, Tolerance := 0.5)
	AND Drive.bIN_STANDSTILL AND Drive.bNEW_VALUE_POSSIBLE  THEN
	DriveVar.Out_InPos := TRUE;
	DriveVar.In_MoveAbs := FALSE;
	DriveVar.In_MoveRel := FALSE;
	ServoBusy := FALSE;
END_IF

IF plsEMGReset.Q AND Drive.bIN_STANDSTILL AND Drive.bIN_REFERENCE AND
	Drive.bNEW_VALUE_POSSIBLE THEN
	DriveVar.Out_InPos := TRUE;
	ServoBusy := FALSE;
END_IF

IF DriveVar.In_StopMove THEN
	DriveVar.In_MoveAbs := FALSE;
	DriveVar.In_MoveHome := FALSE;
	DriveVar.In_MoveRel := FALSE;
	DriveVar.In_JogBwd := FALSE;
	DriveVar.In_JogFwd := FALSE;
	DriveVar.In_StopMove := FALSE;
	(* Stop Movement *)
	Drive.bJOG_FORWARD := TRUE;
	Drive.bJOG_BACKWARD := TRUE;
	ServoBusy := FALSE;

ELSIF 	Drive.bJOG_FORWARD AND Drive.bJOG_BACKWARD AND MC.AutoMode THEN
	Drive.bJOG_FORWARD 	:= FALSE;
	Drive.bJOG_BACKWARD := FALSE;
END_IF


(***********************************************************************************************)
(*Servo Function Block*)
Drive(
	stEK_IN:= In_DriveInput, 
	bSTATUS_MESSAGE=> , 
	bWARNING=> , 
	bERROR=> , 
	dwDRIVE_DIAGNOSIS=> , 
	stEK_OUT=> Out_DriveOutput );

	
	Out_DriveOutput.wSignalsteuerwort.6 := drive.bJOG_FORWARD;
	Out_DriveOutput.wSignalsteuerwort.7 := drive.bJOG_BACKWARD;
	
(***********************************************************************************************)
(*Set Reference Point for Absulute Encoder Servo*)
plsHomed(CLK :=Drive.bIN_REFERENCE);
	
IF In_AbsEncoder THEN
	Out_DriveOutput.wSignalsteuerwort.1 := DriveVar.In_SetAbsRef;
	
	IF Drive.bIN_REFERENCE THEN
		DriveVar.Out_Referenced := TRUE;
	ELSE
		DriveVar.Out_Referenced := FALSE;	
	END_IF
ELSE
	Out_DriveOutput.wSignalsteuerwort.8 := DriveVar.In_SetAbsRef;
	DriveVar.Out_Referenced := In_DriveInput.wSignalstatuswort.2;	
	IF plsHomed.Q THEN
		DriveVar.In_SetAbsRef := FALSE;
	END_IF
END_IF


	
(***********************************************************************************************)
(*Set Station Error Bit if Servo has error*)
tmrMajorErrorRecovery (IN := mc.E_EmgStop OR mc.E_LightCurtain OR mc.E_SafetyDoorOpen OR mc_ctrl.In_OtherTrouble OR Guard_Door.Guard_Door_Fault, pt:=T#2S);

IF tmrMajorErrorRecovery.Q THEN
	DriveVar.Out_ErrorWord	:= 0;
END_IF
IF DriveVar.Out_Error THEN 
	DriveVar.In_MoveAbs	:= FALSE;	
END_IF

Station.DeviceFault := DriveVar.Out_Error OR Station.DeviceFault;

END_FUNCTION_BLOCK

// ---- POUs/FB/fbVacuumValveCtrl.TcPOU
FUNCTION_BLOCK fbVacuumValveCtrl

VAR_INPUT
	IN_Name:				STRING;
	In_Enable:				BOOL;
	In_Reset:				BOOL;


	(*Sensors*)
	In_Vacuum_Switch:		BOOL;
	In_Drop_Monitor_Enable:	BOOL;

	(*Timer*)
	In_VacuumTON:			TIME;
	In_Release_TON:			TIME;
	In_PurgeTON:			TIME;
	in_Timeout:				TIME;
END_VAR

VAR_OUTPUT
	Out_VacuumSV:			BOOL;
	Out_PurgeSV:			BOOL;
END_VAR

VAR

	Loc_Vacuum:				BOOL;
	Loc_Purge:				BOOL;
	Err_Vacuum:				BOOL;
	VAcuum_TOut:			TON;
	Purge_TOut: 				TON;
	Vacuum_TON:			TON;
	Release_TON: 			TON;
	Purge_TON:				TON;
	Purge_ON:				BOOL;
	Loc_VacuumPls: 			BOOL;
	PurgePls:				R_TRIG;
	VacuumPls: 				R_TRIG;
	Loc_PurgePls: 			BOOL;
	Out_RSErr:				BOOL;
	VacuumPosPls: 			F_TRIG;
	PurgePosPls: 			F_TRIG;
	plsManualOff: R_TRIG;
END_VAR
VAR_IN_OUT
	VacVar:structVacuum;
	Station:structStationCtrl;
END_VAR
VAR // added by the converter: edge detectors and wires of the graphical bodies
    _w1, _w2, _w3, _w4, _w5 : BOOL;
END_VAR

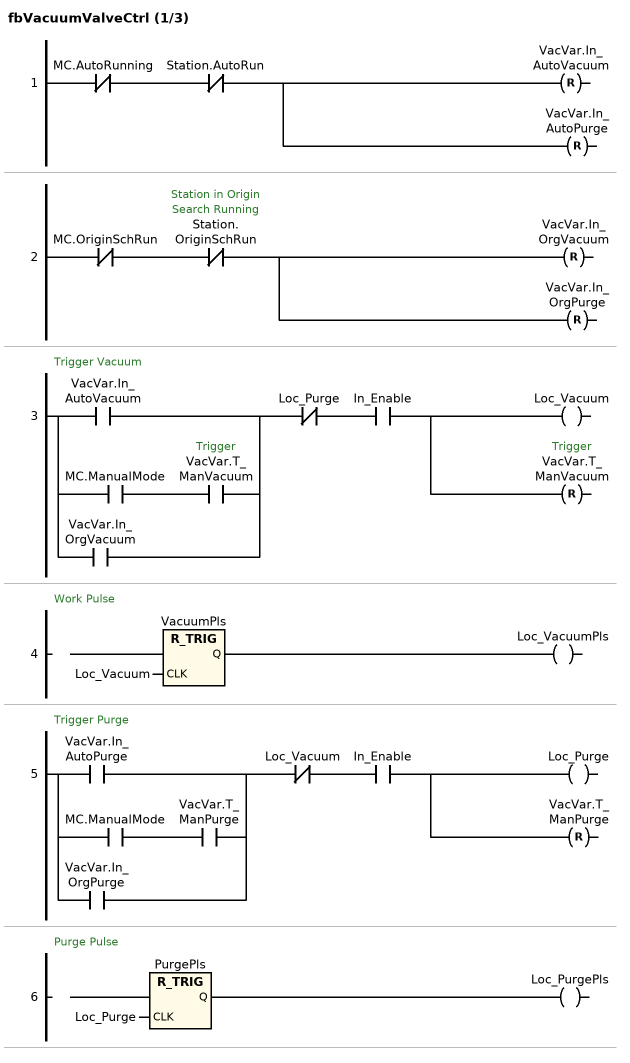
// NETWORK 1
_w1 := NOT MC.AutoRunning AND NOT Station.AutoRun;
VacVar.In_AutoVacuum R= _w1;
VacVar.In_AutoPurge R= _w1;

// NETWORK 2
//   Station.OriginSchRun: Station in Origin Search Running
_w2 := NOT MC.OriginSchRun AND NOT Station.OriginSchRun;
VacVar.In_OrgVacuum R= _w2;
VacVar.In_OrgPurge R= _w2;

// NETWORK 3
// Trigger Vacuum
//   VacVar.T_ManVacuum: Trigger
_w3 := (VacVar.In_AutoVacuum OR MC.ManualMode AND VacVar.T_ManVacuum OR VacVar.In_OrgVacuum) AND NOT Loc_Purge AND In_Enable;
Loc_Vacuum := _w3;
VacVar.T_ManVacuum R= _w3;

// NETWORK 4
// Work Pulse
VacuumPls(CLK := Loc_Vacuum); // R_TRIG
Loc_VacuumPls := VacuumPls.Q;

// NETWORK 5
// Trigger Purge
_w4 := (VacVar.In_AutoPurge OR MC.ManualMode AND VacVar.T_ManPurge OR VacVar.In_OrgPurge) AND NOT Loc_Vacuum AND In_Enable;
Loc_Purge := _w4;
VacVar.T_ManPurge R= _w4;

// NETWORK 6
// Purge Pulse
PurgePls(CLK := Loc_Purge); // R_TRIG
Loc_PurgePls := PurgePls.Q;

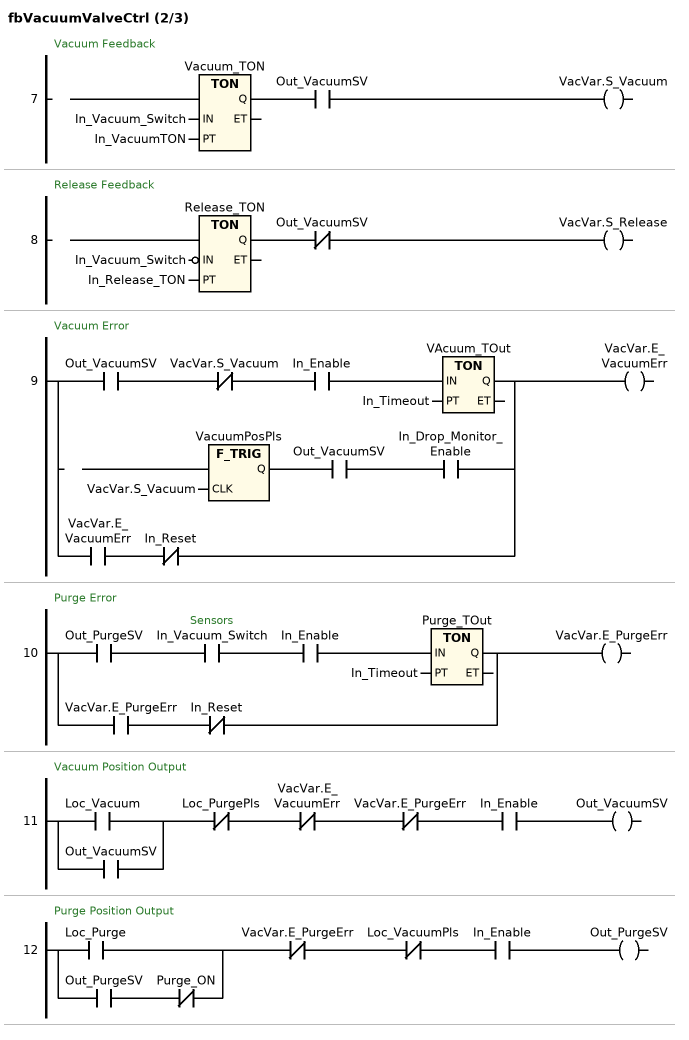
// NETWORK 7
// Vacuum Feedback
//   In_Vacuum_Switch: Sensors
//   In_VacuumTON: Timer
Vacuum_TON(IN := In_Vacuum_Switch, PT := In_VacuumTON); // TON
VacVar.S_Vacuum := Vacuum_TON.Q AND Out_VacuumSV;

// NETWORK 8
// Release Feedback
//   In_Vacuum_Switch: Sensors
Release_TON(IN := NOT In_Vacuum_Switch, PT := In_Release_TON); // TON
VacVar.S_Release := Release_TON.Q AND NOT Out_VacuumSV;

// NETWORK 9
// Vacuum Error
VAcuum_TOut(IN := Out_VacuumSV AND NOT VacVar.S_Vacuum AND In_Enable, PT := In_Timeout); // TON
VacuumPosPls(CLK := VacVar.S_Vacuum); // F_TRIG
VacVar.E_VacuumErr := VAcuum_TOut.Q OR VacuumPosPls.Q AND Out_VacuumSV AND In_Drop_Monitor_Enable OR VacVar.E_VacuumErr AND NOT In_Reset;

// NETWORK 10
// Purge Error
//   In_Vacuum_Switch: Sensors
Purge_TOut(IN := Out_PurgeSV AND In_Vacuum_Switch AND In_Enable, PT := In_Timeout); // TON
VacVar.E_PurgeErr := Purge_TOut.Q OR VacVar.E_PurgeErr AND NOT In_Reset;

// NETWORK 11
// Vacuum Position Output
Out_VacuumSV := (Loc_Vacuum OR Out_VacuumSV) AND NOT Loc_PurgePls AND NOT VacVar.E_VacuumErr AND NOT VacVar.E_PurgeErr AND In_Enable;

// NETWORK 12
// Purge Position Output
Out_PurgeSV := (Loc_Purge OR Out_PurgeSV AND NOT Purge_ON) AND NOT VacVar.E_PurgeErr AND NOT Loc_VacuumPls AND In_Enable;

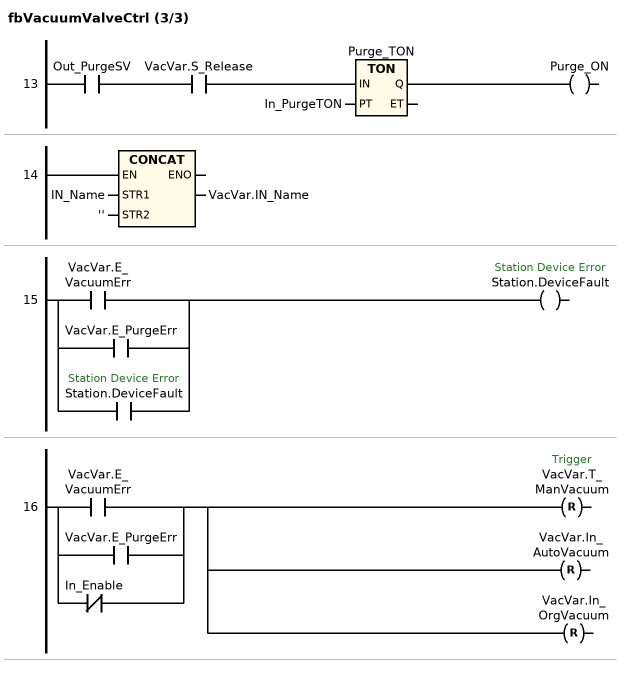
// NETWORK 13
Purge_TON(IN := Out_PurgeSV AND VacVar.S_Release, PT := In_PurgeTON); // TON
Purge_ON := Purge_TON.Q;

// NETWORK 14
VacVar.IN_Name := CONCAT(STR1 := IN_Name, STR2 := '');

// NETWORK 15
//   Station.DeviceFault: Station Device Error
Station.DeviceFault := VacVar.E_VacuumErr OR VacVar.E_PurgeErr OR Station.DeviceFault;

// NETWORK 16
//   VacVar.T_ManVacuum: Trigger
_w5 := VacVar.E_VacuumErr OR VacVar.E_PurgeErr OR NOT In_Enable;
VacVar.T_ManVacuum R= _w5;
VacVar.In_AutoVacuum R= _w5;
VacVar.In_OrgVacuum R= _w5;

END_FUNCTION_BLOCK

// ---- POUs/FB/fbMachineCtrl.TcPOU
FUNCTION_BLOCK fbMachineCtrl

VAR_INPUT
	In_Start_PB:						BOOL;
	In_Stop_PB:							BOOL;
	In_EmgOK:							BOOL;
	In_Door_Sw: 						BOOL;
	In_Pressure_Sw: 					BOOL;
	In_LightCurtainSafeToCross:			BOOL;
	In_LightCurtainOK: 					BOOL;
	In_CommunicationOK:					BOOL;
	In_IncomingPowerPhase_OK:			BOOL;
	In_OtherTrouble: 					BOOL;
	In_Reset_PB:						BOOL;
	In_Start_Enable:					BOOL;
	In_EndProdWPCleared:				BOOL;
	In_WaitingForMaterial:				BOOL;	
	I_StepFwdPB:						BOOL;
	I_StepBwdPB:						BOOL;

END_VAR

VAR_IN_OUT
	McVar:structMachineCtrl;
	HMI:structHMI;
END_VAR

VAR_OUTPUT
	Out_RedTower:BOOL;
	Out_YelTower :BOOL;
	Out_GrnTower:BOOL;
	Out_Buzzer:BOOL;
	Out_StartPL:BOOL;
	Out_StopPL:BOOL;
	Out_ResetPL:BOOL;
	
END_VAR

VAR
	Loop: INT;
	LoopStation: INT;
(*************************************************************************************************************************************)
(*Status Bit*)
(*************************************************************************************************************************************)

	AllStationStop:BOOL;

(*************************************************************************************************************************************)
(*Auto*)
(*************************************************************************************************************************************)
	AutoPBMem	: BOOL;
	StartMem	: BOOL;
	StartDly	: Ton;
	StartCmdHoldDly	:	TON;
	NotAutoRunning:BOOL;

		
	pls_OriginSchRun: R_TRIG;
	OriginSchRunPls: BOOL;

(*************************************************************************************************************************************)
(*Manual*)
(*************************************************************************************************************************************)
	Pls_StepFwd: 	R_TRIG;
	Pls_StepBwd: 	R_TRIG;
	CycleTimer: 	TON;
	ManualCond: 	BOOL;
	T_LampTest:		BOOL;
(*************************************************************************************************************************************)
	(* Error Handling*)
(*************************************************************************************************************************************)
	tmrResetOffDly	:TOF;
	
	tmrEmgOn: TON;
	EmgPBTON :BOOL;

	tmrEmgOn_Air: TON;
	EmgPBTON_Air: BOOL;

	pls_Reset :R_TRIG;
	ResetPls:BOOL;

	tmrDoorSwitch: TON;
	DoorSwTOFF: BOOL;

	tmrCurtainCrossed: TON;
	CurtainCrossedTON:BOOL;


	plsManPBOff: R_trig;
	plsResetCycleTime:ARRAY[1..20] OF r_trig;
	plsResetIdleTime:ARRAY[1..20] OF r_trig;
	plsAutorun:r_trig;
	
END_VAR

(**************************************************************************************************************)
(* Auto Mode Selection*)
(**************************************************************************************************************)
plsManPBOff(CLK:= NOT HMI.T_Manual);

IF (HMI.T_Auto OR plsManPBOff.Q) AND 
	NOT MC.Trouble AND 
	NOT MC.StationStopErr THEN
	AutoPBMem := TRUE;
END_IF;

IF( AutoPBMem OR MC.AutoRunning) AND NOT MC.Trouble THEN
	MC.AutoMode := TRUE;
ELSE
	MC.AutoMode := FALSE;
	AutoPBMem := FALSE;
END_IF;

(**************************************************************************************************************)
(*Manual Mode Selection*)
(**************************************************************************************************************)
IF HMI.T_Manual THEN
	AutoPBMem := FALSE;
END_IF;

IF NOT (AutoPBMem OR MC.AutoRunning) THEN
	MC.ManualMode :=TRUE;
ELSE
	MC.ManualMode :=FALSE;
END_IF;

IF NOT MC.AutoRunning THEN (*Do Not Process during Autorun to Optimize Cyclic Time*)
	
(**************************************************************************************************************)
	(* Manual Interlocking *)
	(**************************************************************************************************************)
	
	ManualSafetyOK 	:= NOT MC.Trouble;
	ManualCond 		:= MC.ManualMode AND ManualSafetyOK AND NOT mc.OriginSchRun;
	
	(**************************************************************************************************************)
	(* Manual General*)
	(**************************************************************************************************************)
	
	Pls_StepFwd(CLK:= I_StepFwdPB OR HMI.T_StepFwd);
	M_StepFwdPls := Pls_StepFwd.Q;
	
	Pls_StepBwd(CLK:= I_StepBwdPB OR HMI.T_StepBwd);
	M_StepBwdPls := Pls_StepBwd.Q;
	
	(**************************************************************************************************************)
	(* Manual Stepping Mode*)
	(**************************************************************************************************************)
	IF (NOT HMI.T_StepStop) AND ManualCond AND
		NOT (SC[HMI.T_Curr_Step_Station].MajorFault OR 
			SC[HMI.T_Curr_Step_Station].MinorFault OR
			SC[HMI.T_Curr_Step_Station].DeviceFault OR 
			MC.Trouble OR MC_Ctrl.In_Stop_PB OR MC_Ctrl.HMI.T_Stop OR
				HMI.T_StepStop  ) THEN
		IF HMI.T_StepRun THEN
			M_StepRun := TRUE;
		END_IF;
	ELSE
		M_StepRun := FALSE;
		HMI.T_StepRun := FALSE;	
		HMI.T_StepStop := FALSE;
	END_IF;

	(* Display Status on Visio*)
	HMI.T_StationError 			:= sc[HMI.T_Curr_Step_Station].MajorFault OR sc[HMI.T_Curr_Step_Station].MinorFault;
	HMI.T_Origin 				:= sc[HMI.T_Curr_Step_Station].Origin;
	HMI.V_StepRunCurrStation 	:= sc[HMI.T_Curr_Step_Station].Name;
	HMI.V_StepRunStatus 		:= sc[HMI.T_Curr_Step_Station].Status;
	HMI.T_StepRunning 			:= sc[HMI.T_Curr_Step_Station].M_Step;
	HMI.T_OriginRunning			:= sc[HMI.T_Curr_Step_Station].OriginSchRun;

	FOR Loop := 0 TO Number_of_Station BY 1 DO
		SC[Loop].M_Step		:= FALSE;
	END_FOR

	IF M_StepRun THEN
		SC[HMI.T_Curr_Step_Station].M_Step	:= TRUE;
	END_IF;

	(* CycleTime Calculation*)
	CycleTimer(IN:=M_StepRun , PT:=t#1100h , Q=> , ET=> );
	
	IF M_StepRun THEN
		HMI.T_ManualCycleTime :=CycleTimer.ET;
	END_IF

	(**************************************************************************************************************)
	(*Station Origin Search Run*)
	(**************************************************************************************************************)
	
	IF mc.ManualMode THEN
		(*Handles Origin Search in Step Mode Page*)
		IF 	NOT SC[HMI.T_Curr_Step_Station].Origin AND
			NOT (SC[HMI.T_Curr_Step_Station].MajorFault OR 
			SC[HMI.T_Curr_Step_Station].MinorFault OR
			SC[HMI.T_Curr_Step_Station].DeviceFault OR 
			MC.Trouble OR MC_Ctrl.In_Stop_PB OR MC_Ctrl.HMI.T_Stop OR
				HMI.T_StepStop  )  THEN
			IF HMI.T_StationOriginSearch THEN		
				SC[HMI.T_Curr_Step_Station].OriginSchRun	:= TRUE;
			END_IF
		ELSE
			SC[HMI.T_Curr_Step_Station].OriginSchRun		:= FALSE;
		END_IF		
		(*Handles Individual Station Origin Search Button*)
		FOR Loop := 0 TO Number_of_Station BY 1 DO
			IF NOT SC[Loop].Origin AND
			NOT (SC[Loop].MajorFault OR 
				SC[Loop].MinorFault OR
				SC[Loop].DeviceFault OR 
				MC.Trouble OR MC_Ctrl.In_Stop_PB OR MC_Ctrl.HMI.T_Stop OR
					HMI.T_StepStop )  THEN
				IF SC[Loop].T_OriginSearch THEN		
					SC[Loop].OriginSchRun	:= TRUE;
				END_IF
			ELSE
				SC[Loop].OriginSchRun	:= FALSE;
			END_IF			
		END_FOR
	ELSE
		FOR Loop := 0 TO Number_of_Station BY 1 DO
			SC[Loop].OriginSchRun	:= FALSE;	
		END_FOR
	END_IF;
	
	(**************************************************************************************************************)
	(*Origin Search Run*)
	(**************************************************************************************************************)
	IF MC.ManualMode AND NOT MC.AllOrigin AND 
		NOT (MC.StationStopErr OR MC.Trouble OR MC.StopPressed OR
			 MC_Ctrl.In_Stop_PB OR MC_Ctrl.HMI.T_Stop)  THEN
		IF HMI.T_OriginSearch THEN
			MC.OriginSchRun  := TRUE;
		END_IF;
	ELSE
		MC.OriginSchRun := FALSE;
	END_IF;

	pls_OriginSchRun(CLK:= MC.OriginSchRun);
	OriginSchRunPls := pls_OriginSchRun.Q;
	
	(**************************************************************************************************************)
	(*Dry Run Mode Selection*)
	(**************************************************************************************************************)
	IF NOT MC.AutoRunning AND HMI.T_DryRun THEN
		MC.DryRun := TRUE;
	ELSE
		MC.DryRun := FALSE;
	END_IF;
	
	IF NOT MC.AutoMode THEN
		HMI.T_EndProd := FALSE;
	END_IF;

	(**************************************************************************************************************)
	(* For programmer Station Bypass - Debug Only*)
	(**************************************************************************************************************)
	FOR Loop := 0 TO Number_of_Station DO
		IF HMI.T_Station_BypassP[Loop] THEN
				SC[Loop].Bypass := TRUE;
		ELSE
			SC[Loop].Bypass := FALSE;
		  END_IF;
	END_FOR
	
END_IF	
	
(**************************************************************************************************************)
(* Machine Start *)
(**************************************************************************************************************)
NotAutoRunning := NOT MC.AutoRunning;

StartDly(IN:= StartMem, PT:=T#3S);
StartCmdHoldDly (IN:= 	(In_Start_PB OR HMI.T_Start) AND
						NOT MC.StationStopErr AND
						NOT (In_Stop_PB OR HMI.T_Stop) AND 
						In_Start_Enable AND 
						MC.AllOrigin,
					PT:= T#1S);		

IF MC.AutoRunning THEN
	HMI.V_AutorunString := 'Running';
ELSE
	HMI.V_AutorunString := 'Auto Mode';
END_IF

IF MC.AutoMode AND NOT MC.Stop THEN
	IF StartCmdHoldDly.Q THEN
		StartMem		:= TRUE;
	ELSIF StartDly.Q THEN
		MC.AutoRunning 	:= TRUE;
	ELSIF (In_Start_PB OR HMI.T_Start) AND NOT MC.AllOrigin THEN	
		HMI.V_AutorunString := 'Machine Not Origin';
	END_IF;
ELSE
	MC.AutoRunning 	:= FALSE;
	StartMem		:= FALSE;
END_IF;

(**************************************************************************************************************)
(* Machine Stop *)
(**************************************************************************************************************)
IF MC.AutoRunning THEN
	IF In_Stop_PB OR HMI.T_Stop OR 
		In_EndProdWPCleared OR MC.StationStopErr THEN
		MC.StopPressed := TRUE;
	END_IF;
ELSE
	MC.StopPressed := FALSE;
END_IF;


IF MC.StopPressed AND AllStationStop THEN
	MC.StopPressed := FALSE;
	MC.Stop:=TRUE;
ELSE
	MC.Stop :=FALSE;	
END_IF;
	
(**************************************************************************************************************)
(* Machine Status *)
(*From Station Status*)
(**************************************************************************************************************)

FOR Loop := 0 TO Number_of_Station BY 1  DO
	IF NOT SC[Loop].Running THEN
		AllStationStop := TRUE;
	ELSE
		AllStationStop := FALSE;
		EXIT;
	END_IF
END_FOR

MC.IdleState := AllStationStop;

FOR Loop := 0 TO Number_of_Station BY 1  DO
	IF SC[Loop].Rdy OR SC[LOOP].BYPASS	THEN
		MC.AllStationRdy := TRUE;
	ELSE
		MC.AllStationRdy := FALSE;
		EXIT;
	END_IF
END_FOR

FOR Loop := 0 TO Number_of_Station BY 1  DO
	IF SC[Loop].NoWP THEN
		MC.AllStationNoWP := TRUE;
	ELSE
		MC.AllStationNoWP := FALSE;
		EXIT;
	END_IF
END_FOR

FOR Loop := 0 TO Number_of_Station BY 1  DO
	IF SC[Loop].Origin OR SC[Loop].Bypass THEN
		MC.AllOrigin:= TRUE;
	ELSE
		MC.AllOrigin := FALSE;
		EXIT;
	END_IF
END_FOR

(*Major Error for Immediate Stop*)
MC.Trouble:=	MC.E_EmgStop OR 
				MC.E_AirLow OR 
				MC.E_LightCurtain OR 
				MC.E_Communication OR 
				MC.E_SafetyDoorOpen OR
				MC.E_IncomingPowerPhase OR
				In_OtherTrouble;

FOR Loop := 0 TO Number_of_Station BY 1  DO
	IF SC[Loop].MajorFault THEN
		MC.Trouble:= TRUE;
	END_IF
END_FOR

(*Minor Error for Stop after one cycle*)
MC.StationStopErr := MC.E_LightCurtain;

FOR Loop := 0 TO Number_of_Station BY 1  DO
	IF SC[Loop].MinorFault AND NOT SC[Loop].Bypass THEN
		MC.StationStopErr:= TRUE;
	END_IF
END_FOR

(**************************************************************************************************************)
(* Auto Msg Alarm Display  *)
(**************************************************************************************************************)

IF MC.E_Communication THEN
	HMI.T_StatusString 		:= 'Machine Ethercat Communication Major Error';
	HMI.T_StatusStringInt	:= 1;
ELSIF mc.E_IncomingPowerPhase THEN
	HMI.T_StatusString 		:= 'Machine Incoming Power Phase Major Error';
	HMI.T_StatusStringInt	:= 2;
ELSIF MC.E_EmgStop THEN
	HMI.T_StatusString 		:= 'Machine Safety Circuit Broke Major Error';
	HMI.T_StatusStringInt	:= 3;
ELSIF MC.E_AirLow THEN
	HMI.T_StatusString 		:= 'Machine Incoming Air Pressure Low Major Error';
	HMI.T_StatusStringInt	:= 4;
ELSIF MC.E_LightCurtain THEN
	HMI.T_StatusString 		:= 'Machine Light Curtain Crossed Major Error';
	HMI.T_StatusStringInt	:= 5;
ELSIF MC.Trouble THEN
	HMI.T_StatusString 		:= 'Machine Major Error';
	HMI.T_StatusStringInt	:= 6;	
ELSIF MC.StationStopErr THEN
	HMI.T_StatusString 		:= 'Machine Station Error';
	HMI.T_StatusStringInt	:= 7;	
ELSIF MC.StopPressed THEN
	HMI.T_StatusString 		:= 'Machine is Stopping Autorun Mode';
	HMI.T_StatusStringInt	:= 8;	
ELSIF MC.AutoRunning THEN
	HMI.T_StatusString 		:= 'Auto Running';
	HMI.T_StatusStringInt	:= 9;	
ELSIF MC.AutoMode THEN
	HMI.T_StatusString 		:= 'Auto Mode';
	HMI.T_StatusStringInt	:= 10;	
ELSIF MC.ManualMode THEN
	HMI.T_StatusString 		:= 'Manual Mode';
	HMI.T_StatusStringInt	:= 11;	
END_IF

(*************************************************************************************************************************************)
(* Reset Error And Warning Memory*)
(*************************************************************************************************************************************)

tmrEmgOn (IN := In_EmgOK, pt := T#1s);
EmgPBTON := tmrEmgOn.Q;

tmrEmgOn_Air (IN := In_EmgOK AND In_Door_Sw, pt := T#3S);
EmgPBTON_Air := tmrEmgOn_Air.Q;

MC.ResetPressed := HMI.T_Reset OR In_Reset_PB OR tmrResetOffDly.Q;
tmrResetOffDly	(IN:= HMI.T_Reset OR In_Reset_PB, PT:= T#3S);

pls_Reset (CLK := MC.ResetPressed);
ResetPls := pls_Reset.Q;

(* Reset Error*)
	IF tmrResetOffDly.Q THEN
	FOR LoopStation := 0 TO Number_of_Station BY 1 DO
		SC[LoopStation].DeviceFault := FALSE;
		FOR Loop := 1 TO 10 BY 1 DO
			ErrorDWord[LoopStation,Loop] :=0;
			WarningDWord[LoopStation,Loop] :=0;
		END_FOR
	END_FOR

			MC.E_EmgStop				:=FALSE;
			MC.E_LightCurtain			:=FALSE;
			MC.E_AirLow 				:=FALSE;
			MC.E_SafetyDoorOpen			:=FALSE;
			MC.E_Communication 			:=FALSE;
			MC.E_IncomingPowerPhase 	:=FALSE;
			
	END_IF;

(* Set Warning*)

MC.Warning := FALSE;
FOR LoopStation := 0 TO Number_of_Station BY 1 DO
	FOR Loop := 1 TO 10 DO
		IF WarningDWord[LoopStation,Loop]>0 OR sc[LoopStation].Warning THEN
			MC.Warning := TRUE;
		END_IF;
	END_FOR
END_FOR

HMI.T_AutoMsgAlarm := MC.Trouble OR MC.StationStopErr OR (NOT MC.AutoRunning AND NOT MC.AllOrigin) ;

(*************************************************************************************************************************************)
(*Error And Warning Summaries*)
(*************************************************************************************************************************************)
MC.ErrDetection := MC.AutoRunning OR MC.OriginSchRun;

(*************************************************************************************************************************************)
(*General Error and Trouble*)
(*************************************************************************************************************************************)

(*Incoming Power Phase Error*)
IF NOT In_IncomingPowerPhase_OK THEN
	MC.E_IncomingPowerPhase	:=TRUE;
END_IF

(*E-stop Error*)

IF NOT EmgPBTON THEN
	MC.E_EmgStop := TRUE;
END_IF;

(*Safety Door Error*)
tmrDoorSwitch (in:= NOT In_Door_Sw, PT:= T#1S);
DoorSwTOFF := tmrDoorSwitch.q;

IF DoorSwTOFF AND NOT HMI.T_BypassDoor THEN
	MC.E_SafetyDoorOpen := TRUE;
END_IF;

(*Air Low Error*)
IF EmgPBTON_Air AND NOT In_Pressure_Sw THEN
	MC.E_AirLow := TRUE;
END_IF;

(*Light Curtain Crossed Error*)
tmrCurtainCrossed(IN := NOT In_LightCurtainOK, PT:= t#0.1s);
CurtainCrossedTON := tmrCurtainCrossed.Q;

IF NOT In_LightCurtainSafeToCross  AND NOT In_LightCurtainOK THEN
	MC.E_LightCurtain := TRUE;
END_IF;

(*Communication Bus Error*)
IF EmgPBTON AND In_CommunicationOK THEN
	MC.E_Communication := TRUE;
END_IF

(**************************************************************************************************************)
(* General Output*)
(**************************************************************************************************************)

Out_RedTower := MC.Trouble OR 
				( MC.StationStopErr AND ON_1s) OR
				(mc.ManualMode AND T_LampTest);

Out_YelTower := MC.ManualMode OR 
				( MC.Warning AND ON_1s AND NOT  MC.Trouble AND NOT  MC.StationStopErr ) OR
				(mc.ManualMode AND T_LampTest);

Out_GrnTower := ((MC.AutoRunning AND NOT MC.StopPressed) OR NOT AllStationStop) OR 
				(MC.StopPressed AND ON_1s) OR
				(mc.ManualMode AND T_LampTest);

IF NOT (Out_RedTower OR MC.Warning) THEN
	HMI.T_BuzzerOff := FALSE;
END_IF

Out_Buzzer := 	(Out_RedTower OR (MC.Warning AND ON_1s) OR 
				(mc.ManualMode AND T_LampTest) OR
				(StartMem AND NOT MC.AutoRunning AND ON_50ms)) AND NOT HMI.T_BuzzerOff AND NOT HMI.T_BypassBuzzer;

Out_StartPL := 	(((*MC.AutoRunning AND In_WaitingForMaterial) OR*) MC.StopPressed (*OR StartMem*)) AND ON_1s) OR
				(mc.ManualMode AND T_LampTest) OR
			(mc.AutoMode AND NOT (*MC.StationStopErr*) mc.AutoRunning AND
				NOT (In_Stop_PB OR HMI.T_Stop) AND 
				NOT W_ServiceStop AND
					In_Start_Enable AND 
					MC.AllOrigin);

Out_StopPL 	:= 	(MC.StopPressed AND ON_1s) OR (NOT MC.AutoRunning);

Out_ResetPL := 	(MC.Trouble OR MC.StationStopErr) OR
				(mc.ManualMode AND T_LampTest) OR
				MC.StopPressed OR
				W_ServiceStop;			

(**************************************************************************************************************)
(* Station Cylce Time Calculation*)
(**************************************************************************************************************)

FOR LoopStation := 0 TO Number_of_Station BY 1 DO
	plsResetCycleTime[LoopStation] (CLK := SC[LoopStation].Running);
	IF plsResetCycleTime[LoopStation].Q THEN
		IF MC.AutoMode THEN
			IF SC[LoopStation].CycleTimeSecAvg > 0 THEN
				SC[LoopStation].CycleTimeSecAvg := (SC[LoopStation].CycleTimeSecAvg+SC[LoopStation].CycleTimeSec)/2;
			ELSE
				SC[LoopStation].CycleTimeSecAvg := SC[LoopStation].CycleTimeSec;
			END_IF
		END_IF
		SC[LoopStation].CycleTimeSec := 0;
	END_IF
	
	plsResetIdleTime[LoopStation] (CLK := SC[LoopStation].AutoRun AND NOT SC[LoopStation].Running);
	IF plsResetIdleTime[LoopStation].Q THEN
		IF MC.AutoMode THEN
			IF SC[LoopStation].IdleTimeSecAvg > 0 THEN
				SC[LoopStation].IdleTimeSecAvg := (SC[LoopStation].IdleTimeSecAvg+SC[LoopStation].IdleTimeSec)/2;
			ELSE
				SC[LoopStation].IdleTimeSecAvg := SC[LoopStation].IdleTimeSec;
			END_IF
		END_IF
		SC[LoopStation].IdleTimeSec := 0;
	END_IF
	
	IF SC[LoopStation].Running AND
		Clock100msOnPls THEN
		SC[LoopStation].CycleTimeSec := SC[LoopStation].CycleTimeSec + 0.1 ;
	ELSIF SC[LoopStation].AutoRun AND NOT SC[LoopStation].Running AND
		Clock100msOnPls THEN
		SC[LoopStation].IdleTimeSec := SC[LoopStation].IdleTimeSec + 0.1 ;
	END_IF
END_FOR

END_FUNCTION_BLOCK

// ---- POUs/Collator/CO_Motor_Output.TcPOU
PROGRAM CO_Motor_Output
VAR
	Reset:BOOL;
		
	plsStackRelWork: R_trig;
	plsStackRelHome: R_trig;
	tmrStackRelHome: Ton;
	tmrPresserHold:TOF;
	
	StackStopMem	:BOOL;
	tmrStackStopDly	:Ton;
	
END_VAR


CO_Cv_Mtr_Var.In_MoveXLock := TRUE;
IF HMI.V_MachineSpeed <25 THEN
	CO_Cv_Mtr_Var.In_SpeedSel  := 0;
ELSIF HMI.V_MachineSpeed >=25 AND HMI.V_MachineSpeed <50  THEN
	CO_Cv_Mtr_Var.In_SpeedSel  := 1;
ELSIF HMI.V_MachineSpeed >=50 AND HMI.V_MachineSpeed <75  THEN
	CO_Cv_Mtr_Var.In_SpeedSel  := 2;	
ELSIF HMI.V_MachineSpeed >=75 THEN
	CO_Cv_Mtr_Var.In_SpeedSel  := 3;
END_IF;

CO_Cv_Mtr(
	IN_DevName:= 'COLLATOR INFEED CV', 
	In_Enable:= TRUE, 
	In_Reset:= MC.ResetPressed, 
	In_InvRdy := I_CO_Cv_InvRdy, 
	Out_InvRun => O_CO_CV_Mtr_Run, 
	Out_InvDirc => O_CO_CV_Mtr_Dirc, 
	Out_InvSpdBit0 => O_CO_CV_Mtr_Spd1, 
	Out_InvSpdBit1 => O_CO_CV_Mtr_Spd2, 
	MotorVar:= CO_Cv_Mtr_Var,
	Station			:= SC[0]);

//***************************************************************************************

CO_UpStreamCv_Mtr_Var.In_MoveXLock	:= TRUE;
	
CO_UpStreamCv_Mtr(
	IN_DevName:= 'COLLATOR UPSTREAM CV', 
	In_Enable:= Cfg_Upstream_Conveyor, 
	In_Reset:= MC.ResetPressed, 
	In_InvRdy := I_UpStreamInfeedRdy	, 
	Out_InvRun => O_UpStreamInfeedCv, 
	Out_InvDirc => , 
	Out_InvSpdBit0 => , 
	Out_InvSpdBit1 => , 
	MotorVar:= CO_UpStreamCv_Mtr_Var,
	Station			:= SC[0]);	
	

//**********************************************************************************

tmr_CoStkMtrStop(IN:= I_CO_Stk_Mtr_HomePos, PT:= T#5MS);
pls_CoStkMtrStop(CLK:= tmr_CoStkMtrStop.Q);

IF I_CO_Stk_Mtr_UpPos AND O_CO_Stk_Mtr_Run THEN
	StackStopMem := TRUE;
END_IF

tmrStackStopDly(IN:= StackStopMem , PT:= T#300MS);

IF tmrStackStopDly.Q OR (StackStopMem AND I_CO_Stk_Mtr_HomePos)  THEN
	CO_Stk_Mtr_Var.T_ManOff 	:= TRUE;
	CO_Stk_Mtr_Var.T_ManOn		:= FALSE;
	CO_Stk_Mtr_Var.In_AutoON 	:= FALSE;
	CO_Stk_Mtr_Var.In_OrgOn		:= FALSE;
	StackStopMem				:= FALSE;
ELSIF NOT O_CO_Stk_Mtr_Run THEN
	CO_Stk_Mtr_Var.T_ManOff := FALSE;
END_IF	
CO_Stk_Mtr_Var.In_MoveXLock := I_CO_Bdl_DoorSwitch;

(*
(*================== Option for Non CAM stacker =============================*)
tmrPresserHold(IN:= I_CO_Stk_Mtr_UpPos AND O_CO_Stk_Mtr_Run  , PT:=T#0.1S , Q=> , ET=> );
O_CO_HolderON	:= tmrPresserHold.Q;
*)
CO_Stk_Mtr_Var.In_SpeedSel  := 3;
	
CO_Stk_Mtr(
	IN_DevName:= 'STACKING CAM', 
	In_Enable:= TRUE, 
	In_Reset:= MC.ResetPressed, 
	In_InvRdy := I_CO_Stk_InvRdy, 
	Out_InvRun => O_CO_Stk_Mtr_Run, 
	Out_InvDirc => O_CO_Stk_Mtr_Dirc, 
	Out_InvSpdBit0 => O_CO_Stk_Mtr_Spd1, 
	Out_InvSpdBit1 => O_CO_Stk_Mtr_Spd2, 
	MotorVar:= CO_Stk_Mtr_Var,
	Station			:= SC[0]);
	
IF NOT O_CO_Stk_Mtr_Run AND I_CO_Stk_Mtr_HomePos THEN	
O_CO_Stk_Mtr_ClutchBrake :=	FALSE;
END_IF

IF O_CO_Stk_Mtr_Run THEN
O_CO_Stk_Mtr_ClutchBrake :=	TRUE;	
END_IF












(*
IF ER.AutoRun OR EL.AutoRun OR
	ER.M_Step OR EL.M_Step OR
	MC.AutoMode THEN
	ER_VacPump_Mtr_Var.In_AutoON := TRUE;
ELSE
	ER_VacPump_Mtr_Var.In_AutoON := FALSE;
END_IF

ER_VacPump_Mtr_Var.In_MoveXLock := TRUE;

ER_VacPump_Mtr(
	IN_DevName:= 'VACUUM PUMP', 
	In_Enable:= TRUE, 
	In_Reset:= MC.ResetPressed, 
	In_StarterOK:= I_VacPump_OK, 
	Out_MotorOn=> O_VacPump_On, 
	MotorVar:= ER_VacPump_Mtr_Var,
	Station			:= SC[0]);	
*)	
(*	
CO_Brake_Clutch_Var.In_MoveXLock := TRUE;

CO_Brake_Clutch(
	IN_DevName:= 'BRAKE CLUTCH', 
	In_Enable:= TRUE, 
	In_Reset:= MC.ResetPressed, 
	In_StarterOK:= TRUE, 
	Out_MotorOn=> O_CO_Stk_Mtr_ClutchBrake, 
	MotorVar:= CO_Brake_Clutch_Var,
	Station			:= SC[0]);		
*)

END_PROGRAM

// ---- POUs/Collator/CO_TestServo.TcPOU
PROGRAM CO_TestServo
VAR
	plsTestSequence: R_trig;
	TestSequencePosX1: REAL;
	TestSequencePosX2: REAL;
	TestSequencePosY1: REAL;
	TestSequencePosY2: REAL;
	TestSequenceInPos: Ton;
	TestSequenceStep: INT;
	TestBit:BOOL;
	
END_VAR

(*Test Servo Sequence*)
IF MC.ManualMode AND NOT MC.Trouble AND 
	(CO_XPush_Srv_Var.In_MoveXLock OR
	CO_YPush_Srv_Var.In_MoveXLock) AND 
	TestBit THEN
	IF HMI.T_Start AND
		(CO_XPush_Srv_Var.In_MoveXLock AND
		CO_YPush_Srv_Var.In_MoveXLock) THEN
		TestSequence := TRUE;
		CO_XPush_Srv_Var.In_ServoOn := TRUE;
		CO_YPush_Srv_Var.In_ServoOn := TRUE;
		TestSequenceStep := 10;
	END_IF
	IF HMI.T_Stop THEN
		TestSequence := FALSE;
		TestSequenceStep := 0;
	END_IF
ELSE
	TestSequence := FALSE;
	TestSequenceStep := 0;
END_IF

plsTestSequence(CLK:=TestSequence);

TestSequenceInPos (IN := CO_XPush_Srv_Var.Out_InPos AND
							CO_YPush_Srv_Var.Out_InPos, pt := T#0.1S);

IF TestSequence THEN

	CO_XPush_Srv_Var.In_VelCmd := 1800000;
	CO_YPush_Srv_Var.In_VelCmd := 1800000;
	TestSequencePosX1 := 200;
	TestSequencePosX2 := 1100;
	TestSequencePosY1 := 100;
	TestSequencePosY2 := 1000;
	
	CASE TestSequenceStep OF
		10:
			IF CO_XPush_Srv_Var.Out_Ready THEN
				CO_XPush_Srv_Var.In_PosCmd := TestSequencePosX1;
				CO_XPush_Srv_Var.In_MoveAbs := TRUE;				
			END_IF
			IF CO_YPush_Srv_Var.Out_Ready THEN
				CO_YPush_Srv_Var.In_PosCmd := TestSequencePosY1;
				CO_YPush_Srv_Var.In_MoveAbs := TRUE;				
			END_IF

			IF fcComparePos(CurrPos:= CO_XPush_Srv_Var.Out_CurrPos, TargetPos:= TestSequencePosX1) AND
				fcComparePos(CurrPos:= CO_YPush_Srv_Var.Out_CurrPos, TargetPos:= TestSequencePosY1) THEN
				EL_Srv_Var.In_MoveAbs := FALSE;
				TestSequenceStep := TestSequenceStep + 10;
			END_IF
			
		20:
			IF TestSequenceInPos.Q THEN
				TestSequenceStep := TestSequenceStep + 10;
			END_IF
			
		30:
			IF CO_XPush_Srv_Var.Out_Ready THEN
				CO_XPush_Srv_Var.In_PosCmd := TestSequencePosX2;
				CO_XPush_Srv_Var.In_MoveAbs := TRUE;
			END_IF
			IF CO_YPush_Srv_Var.Out_Ready THEN
				CO_YPush_Srv_Var.In_PosCmd := TestSequencePosY2;
				CO_YPush_Srv_Var.In_MoveAbs := TRUE;
			END_IF
				
			IF fcComparePos(CurrPos:= CO_XPush_Srv_Var.Out_CurrPos, TargetPos:= TestSequencePosX2) AND
				fcComparePos(CurrPos:= CO_YPush_Srv_Var.Out_CurrPos, TargetPos:= TestSequencePosY2) THEN
				EL_Srv_Var.In_MoveAbs := FALSE;
				TestSequenceStep := TestSequenceStep + 10;
			END_IF

		40:
			IF TestSequenceInPos.Q THEN
				TestSequenceStep := 10;
			END_IF
		
	END_CASE
ELSE
	TestSequenceStep := 0;	
END_IF

END_PROGRAM

// ---- POUs/FastTask/CO_StkRel_Cyl_FastOutput.TcPOU
PROGRAM CO_StkRel_Cyl_FastOutput
VAR
	plsStackRelWork: R_trig;
	plsStackRelHome: R_trig;
	tmrStackRelHome: Ton;
END_VAR

plsStackRelWork(CLK:=I_CO_Bdl_StackRel_PE2 AND O_CO_Stk_Mtr_Run);
tmrStackRelHome(IN:= O_CO_StkRel_Bwd, PT:= T#150MS);
plsStackRelHome(CLK:= I_CO_Stk_UpPos2);
tmr_CoStkMtrStop(IN:= I_CO_Stk_UpPos2, PT:= T#20MS);
pls_CoStkMtrStop(CLK:= tmr_CoStkMtrStop.Q);

IF pls_CoStkMtrStop.Q THEN
	CO_Stk_Mtr_Var.T_ManOff := TRUE;
	CO_Stk_Mtr_Var.In_AutoON := FALSE;
ELSIF NOT O_CO_Stk_Mtr_Run THEN
	CO_Stk_Mtr_Var.T_ManOff := FALSE;
END_IF

(*
(* Control Stack Release Cylinder Immediate Response to avoid bundle collision*) 
(*IF NOT I_CO_Stk_DnPos THEN*)
	IF plsStackRelWork.Q THEN	(*Retract Cylinder to allow bundle stack up*)
		IF (MC.OriginSchRun OR SC[0].OriginSchRun) THEN
			CO_StkRel_Cyl_Var.In_OrgWork := TRUE;
			CO_StkRel_Cyl_Var.In_OrgHome := FALSE;
		ELSIF SC[0].AutoRun OR SC[0].M_Step THEN
			CO_StkRel_Cyl_Var.In_AutoWork := TRUE;
			CO_StkRel_Cyl_Var.In_AutoHome := FALSE;	
		ELSE
			CO_StkRel_Cyl_Var.T_ManWork := TRUE;
			CO_StkRel_Cyl_Var.T_ManHome := FALSE;			
		END_IF
	ELSIF plsStackRelHome.Q OR MC.OriginSchRun OR SC[0].OriginSchRun OR
		SC[0].RunStep > 40 THEN	(*Extend Cylinder to hold bundle stack*)
		IF (MC.OriginSchRun OR SC[0].OriginSchRun) THEN
			CO_StkRel_Cyl_Var.In_OrgWork := FALSE;
			CO_StkRel_Cyl_Var.In_OrgHome := TRUE;
		ELSIF SC[0].AutoRun OR SC[0].M_Step THEN
			CO_StkRel_Cyl_Var.In_AutoWork := FALSE;
			CO_StkRel_Cyl_Var.In_AutoHome := TRUE;	
		ELSE
			CO_StkRel_Cyl_Var.T_ManWork := FALSE;
			CO_StkRel_Cyl_Var.T_ManHome := TRUE;			
		END_IF
	END_IF
(*END_IF*)

CO_StkRel_Cyl_Var.In_HomeXLock := TRUE (* NOT I_CO_Bdl_StackRel_PE  debug*);
CO_StkRel_Cyl_Var.In_WorkXLock := true (* NOT I_CO_Bdl_Stack_PE OR I_CO_Stk_UpPos debug*);

CO_StkRel_Cyl(
	IN_CylName		:='2Y2 COL. CV STACK RELEASE', 
	In_Enable		:= NOT MC.Trouble AND FALSE (*debug*), 
	In_Reset		:= MC.ResetPressed, 
	In_WorkRS		:= I_CO_FxStkRel_Bwd AND I_CO_MvStkRel_Bwd, 	
	In_HomeRS		:= I_CO_FxStkRel_Fwd AND I_CO_MvStkRel_Fwd, 
	In_WorkTON		:= T#0MS, 
	In_HomeTON		:= T#0MS, 
	in_Timeout		:= TP_Cyl_Timeout, 
	Out_WorkSV		=> O_CO_StkRel_Bwd, 
	Out_HomeSV		=> O_CO_StkRel_Fwd, 
	CylVar			:= CO_StkRel_Cyl_Var,
	Station			:= SC[0]);
	

*)

END_PROGRAM

// ---- POUs/FastTask/FastTask_Main.TcPOU
PROGRAM FastTask_Main
VAR
END_VAR


CO_BdlCount_Auto();

CO_StkRel_Cyl_FastOutput();

END_PROGRAM

// ---- POUs/Horizontal/Downstream_Conveyor.TcPOU
PROGRAM Downstream_Conveyor
VAR
END_VAR


O_DnStream_ReqToStpNO	:= O_UpStream_ReqToStpNC;
O_DnStream_ReqToStpNC	:= O_UpStream_ReqToStpNO;

O_DnStream_Reject		:= Exit_Case_NG;

END_PROGRAM

// ---- GlobalTextList.TcGTLO
TEXTLIST GlobalTextList
  32 = ' '
  24 = ' %s'
  35 = '%i'
  36 = '%s'
  56 = '****'
  18 = '0.0'
  41 = 'Bwd'
  49 = 'Cancel'
  10 = 'Current Pos:'
  17 = 'Current Position:'
  55 = 'Enter Password:'
  3 = 'Error'
  7 = 'Error Message based on text list'
  2 = 'Errpr'
  42 = 'Fwd'
  25 = 'Home'
  33 = 'Input Monitor'
  1 = 'Jog Bwd'
  0 = 'Jog Fwd'
  54 = 'Maintenance'
  27 = 'Mechanical Interlock'
  6 = 'Negative Limit'
  50 = 'New Password1:'
  51 = 'New Password2:'
  29 = 'OFF'
  48 = 'OK'
  47 = 'Old Password:'
  28 = 'ON'
  39 = 'One Cycle'
  52 = 'Operator'
  45 = 'Origin'
  34 = 'Output Monitor'
  5 = 'Positive Limit'
  4 = 'Referenced'
  30 = 'Release'
  22 = 'Reset'
  38 = 'Run'
  44 = 'Running'
  12 = 'Servo Motor Cont'
  14 = 'Servo Motor Control'
  13 = 'Servo Motor Controller'
  21 = 'Servo On'
  8 = 'Start'
  19 = 'Start Absolute'
  20 = 'Start Relative'
  46 = 'Station Error'
  37 = 'Station Select'
  43 = 'Station Status'
  40 = 'Step Control'
  9 = 'Stop'
  23 = 'Stop Move'
  53 = 'Supervisor'
  11 = 'Target Pos:'
  16 = 'Target Position:'
  15 = 'Target Velocity:'
  31 = 'Vacuum'
  26 = 'Work'
END_TEXTLIST

// ---- VISUs/FB/Std_Cylinder_Ctrl.TcVIS
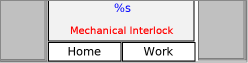
VISUALIZATION Std_Cylinder_Ctrl  // 248x63
VAR_IN_OUT
	m_Input_Inst : None;
END_VAR
    RoundedRectangle (48,0 146x41), "%s", text variable: m_Input_Inst.IN_CylName
    RoundedRectangle (48,42 73x19), "Home", colour toggle: (m_Input_Inst.S_HomePos) <> 0, invisible if: (m_Input_Inst.E_HomeErr) <> 0
    RoundedRectangle (122,42 73x19), "Work", colour toggle: (m_Input_Inst.S_WorkPos) <> 0, invisible if: (m_Input_Inst.E_WorkErr) <> 0
    Group (-1,0 46x59)
        tap m_Input_Inst.T_ManHome
        Button (0,0 48x61)
            tap m_Input_Inst.In_ManHome
        Polygon (38,51)
        Polygon (35,51)
    Group (198,0 46x59)
        tap m_Input_Inst.T_ManWork
        Button (0,0 48x60)
            tap m_Input_Inst.In_ManWork
        Polygon (10,50)
        Polygon (13,50)
    RoundedRectangle (49,21 146x19), "Mechanical Interlock", invisible if: (NOT (NOT m_Input_Inst.In_WorkXLock AND m_Input_Inst.T_ManWork)) <> 0
    RoundedRectangle (49,21 146x19), "Mechanical Interlock", invisible if: (NOT (NOT m_Input_Inst.In_HomeXLock AND m_Input_Inst.T_ManHome)) <> 0
    RoundedRectangle (48,42 73x19), "Home", colour toggle: (m_Input_Inst.E_HomeErr) <> 0, invisible if: (NOT m_Input_Inst.E_HomeErr) <> 0
    RoundedRectangle (122,42 73x19), "Work", colour toggle: (m_Input_Inst.E_WorkErr) <> 0, invisible if: (NOT m_Input_Inst.E_WorkErr) <> 0
END_VISUALIZATION

// ---- VISUs/FB/Std_OnOffDev_Ctrl.TcVIS
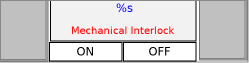
VISUALIZATION Std_OnOffDev_Ctrl  // 249x63
VAR_IN_OUT
	m_Input_Inst : None;
END_VAR
    RoundedRectangle (50,0 146x41), "%s", text variable: m_Input_Inst.IN_DevName
    RoundedRectangle (49,42 73x19), "ON", colour toggle: (m_Input_Inst.S_OnSig) <> 0
    RoundedRectangle (123,42 73x19), "OFF", colour toggle: (NOT m_Input_Inst.S_OnSig) <> 0
    RoundedRectangle (50,21 146x19), "Mechanical Interlock", invisible if: (NOT (NOT m_Input_Inst.In_OnXLock AND m_Input_Inst.T_ManOn)) <> 0
    Group (0,0 46x59)
        tap m_Input_Inst.T_ManOn
        Button (0,0 48x61)
        Polygon (38,51)
        Polygon (35,51)
    Group (199,0 46x59)
        tap m_Input_Inst.T_ManOff
        Button (0,0 48x60)
        Polygon (10,50)
        Polygon (13,50)
END_VISUALIZATION

// ---- VISUs/FB/Std_VacuumVal_Ctrl.TcVIS
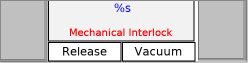
VISUALIZATION Std_VacuumVal_Ctrl  // 248x63
VAR_IN_OUT
	m_Input_Inst : None;
END_VAR
    RoundedRectangle (48,0 146x41), "%s", text variable: m_Input_Inst.IN_Name
    RoundedRectangle (48,42 73x19), "Release", colour toggle: (m_Input_Inst.S_Release) <> 0, invisible if: (m_Input_Inst.E_PurgeErr) <> 0
    RoundedRectangle (122,42 73x19), "Vacuum", colour toggle: (m_Input_Inst.S_Vacuum) <> 0, invisible if: (m_Input_Inst.E_VacuumErr) <> 0
    Group (-1,0 46x59)
        tap m_Input_Inst.T_ManPurge
        Button (0,0 48x61)
            tap m_Input_Inst.In_ManHome
        Polygon (38,51)
        Polygon (35,51)
    Group (198,0 46x59)
        tap m_Input_Inst.T_ManVacuum
        Button (0,0 48x60)
            tap m_Input_Inst.In_ManWork
        Polygon (10,50)
        Polygon (13,50)
    RoundedRectangle (48,23 146x19), "Mechanical Interlock", invisible if: (NOT (NOT m_Input_Inst.In_VacuumX AND m_Input_Inst.T_ManVacuum)) <> 0
    RoundedRectangle (48,23 146x19), "Mechanical Interlock", invisible if: (NOT (NOT m_Input_Inst.In_PurgeX AND m_Input_Inst.T_ManPurge)) <> 0
    RoundedRectangle (48,42 73x19), "Release", colour toggle: (m_Input_Inst.E_PurgeErr) <> 0, invisible if: (NOT m_Input_Inst.E_PurgeErr) <> 0
    RoundedRectangle (122,42 73x19), "Vacuum", colour toggle: (m_Input_Inst.E_VacuumErr) <> 0, invisible if: (NOT m_Input_Inst.E_VacuumErr) <> 0
END_VISUALIZATION

// ---- VISUs/FB/Std_BoschServo_Ctrl.TcVIS
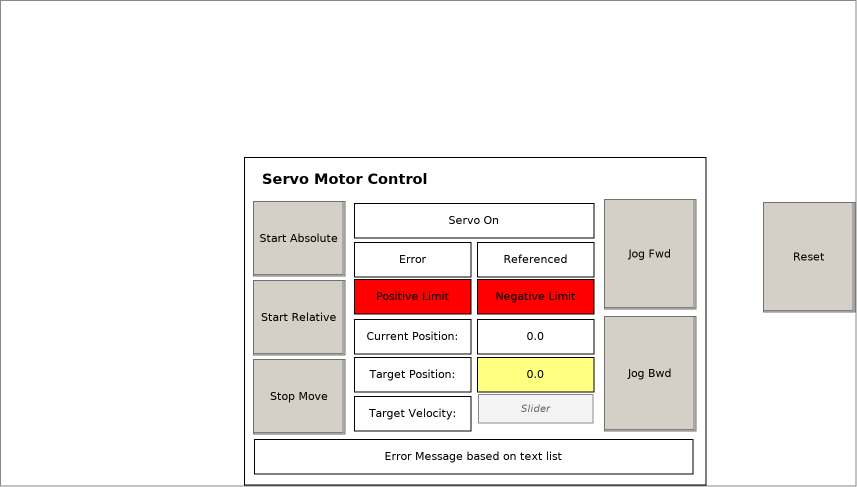
VISUALIZATION Std_BoschServo_Ctrl  // 857x487
    Rectangle (244,157 462x328)
    Button (604,199 92x110), "Jog Fwd"
        tap ER_Arm_Srv_Var.In_JogFwd
    Rectangle (354,242 117x35), "Error", colour toggle: ER_Arm_Srv_Var.Out_Error
    Rectangle (477,242 117x35), "Referenced", colour toggle: ER_Arm_Srv_Var.Out_Referenced
    Rectangle (354,279 117x35), "Positive Limit", colour toggle: ER_Arm_Srv_Var.Out_PosLimit
    Rectangle (477,279 117x35), "Negative Limit", colour toggle: ER_Arm_Srv_Var.Out_NegLimit
    Rectangle (254,439 439x35), "Error Message based on text list", text variable: MAIN.Drive1Var.Out_ErrorWord, colour toggle: ER_Arm_Srv_Var.Out_Error
    Button (604,316 92x115), "Jog Bwd"
        tap ER_Arm_Srv_Var.In_JogBwd
    Button (253,201 92x75), "Start Absolute"
        tap ER_Arm_Srv_Var.In_MoveAbs
    Rectangle (354,319 117x35), "Current Position:"
    Rectangle (354,357 117x35), "Target Position:"
    Rectangle (354,396 117x35), "Target Velocity:"
    Label (259,164 247x30), "Servo Motor Control"
    Rectangle (477,319 117x35), "0.0", text variable: MAIN.Drive1Var.Out_CurrPos, input disabled if: TRUE
    Rectangle (477,357 117x35), "0.0"
    Button (253,280 92x75), "Start Relative"
        tap ER_Arm_Srv_Var.In_MoveRel
    Rectangle (354,203 240x35), "Servo On", colour toggle: ER_Arm_Srv_Var.Out_Ready
        toggle ER_Arm_Srv_Var.In_ServoOn
    Button (763,202 92x110), "Reset"
        tap ER_Servo_Output.Reset
    Button (253,359 92x75), "Stop Move"
        tap ER_Arm_Srv_Var.In_StopMove
    Slider (478,394 115x29), variable: MAIN.Drive1Var.In_VelCmd, scale 0..200
END_VISUALIZATION

// ---- VISUs/Obj_Button/ButtonGreenInd.TcVIS
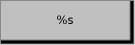
VISUALIZATION ButtonGreenInd  // 135x45
VAR_IN_OUT
	m_Input_ValueTag : None;
END_VAR
VAR_IN_OUT
	m_Input_AssignValue : None;
END_VAR
VAR_IN_OUT
	m_Input_Text : None;
END_VAR
VAR_IN_OUT
	m_Input_ColourTag : None;
END_VAR
VAR_IN_OUT
	m_Input_TapTag : None;
END_VAR
    Rectangle (1,1 132x42)
    Rectangle (0,0 130x40), "%s", text variable: m_Input_Text, colour toggle: (m_Input_ColourTag) <> 0
        tap m_Input_TapTag
        OnMouseUp: execute { m_Input_ValueTag:=(m_Input_AssignValue); }
END_VISUALIZATION

// ---- VISUs/Obj_Indicator/Blue_Ind.TcVIS
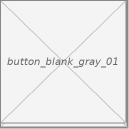
VISUALIZATION Blue_Ind  // 129x129
VAR_IN_OUT
	m_Input_Inst : None;
END_VAR
    Image (0,0 127x127), invisible if: (NOT m_Input_Inst) <> 0, image: button_blank_blue_01
    Image (0,0 126x123), invisible if: (m_Input_Inst) <> 0, image: button_blank_gray_01
END_VISUALIZATION

// ---- VISUs/Obj_Indicator/Green_Ind.TcVIS
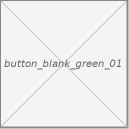
VISUALIZATION Green_Ind  // 129x129
VAR_INPUT
	m_Input_Inst : Bool;
END_VAR
    Image (0,0 127x127), invisible if: (m_Input_Inst) <> 0, image: button_blank_gray_01
    Image (0,0 127x127), invisible if: (NOT m_Input_Inst) <> 0, image: button_blank_green_01
END_VISUALIZATION

// ---- VISUs/Obj_Indicator/Red_Ind.TcVIS
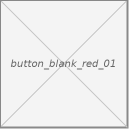
VISUALIZATION Red_Ind  // 129x129
VAR_INPUT
	m_Input_Inst : Bool;
END_VAR
    Image (0,0 127x127), invisible if: (m_Input_Inst) <> 0, image: button_blank_gray_01
    Image (0,0 127x127), invisible if: (NOT m_Input_Inst) <> 0, image: button_blank_red_01
END_VISUALIZATION

// ---- VISUs/Obj_Indicator/Yellow_Ind.TcVIS
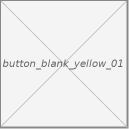
VISUALIZATION Yellow_Ind  // 129x129
VAR_IN_OUT
	m_Input_Inst : None;
END_VAR
    Image (0,0 127x127), invisible if: (m_Input_Inst) <> 0, image: button_blank_gray_01
    Image (0,0 127x127), invisible if: (NOT m_Input_Inst) <> 0, image: button_blank_yellow_01
END_VISUALIZATION

// ---- VISUs/Obj_Switch/ToggleSwitch1.TcVIS
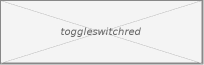
VISUALIZATION ToggleSwitch1  // 204x65
VAR_IN_OUT
	m_Input_Inst : None;
END_VAR
    Image (0,0 202x62), invisible if: (NOT m_Input_Inst) <> 0, image: toggleswitchgreen
        toggle m_Input_Inst
    Image (0,0 202x63), invisible if: (m_Input_Inst) <> 0, image: toggleswitchred
        toggle m_Input_Inst
END_VISUALIZATION

// ---- VISUs/Prog/IO_Monitor.TcVIS
